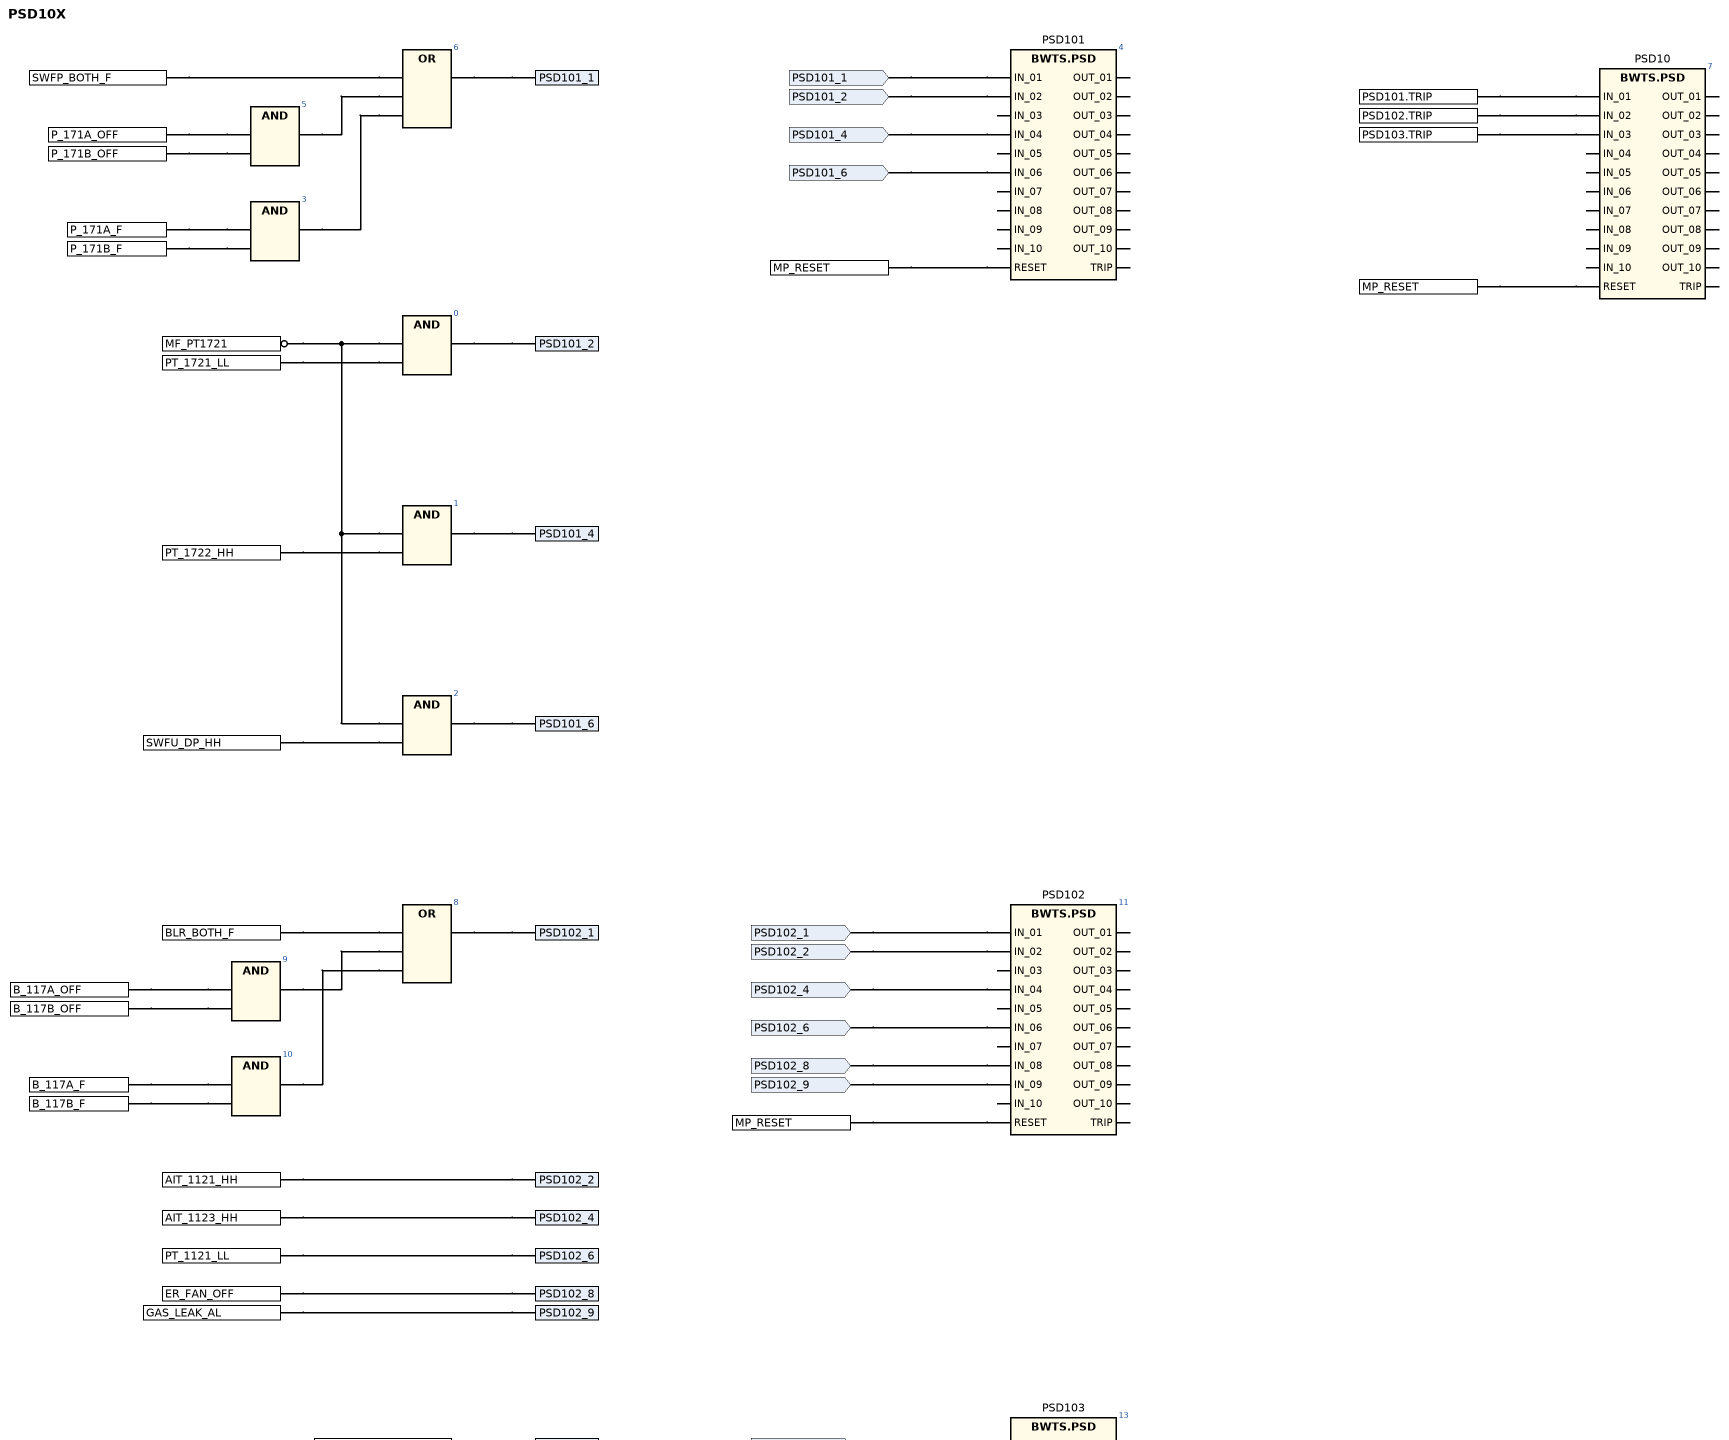
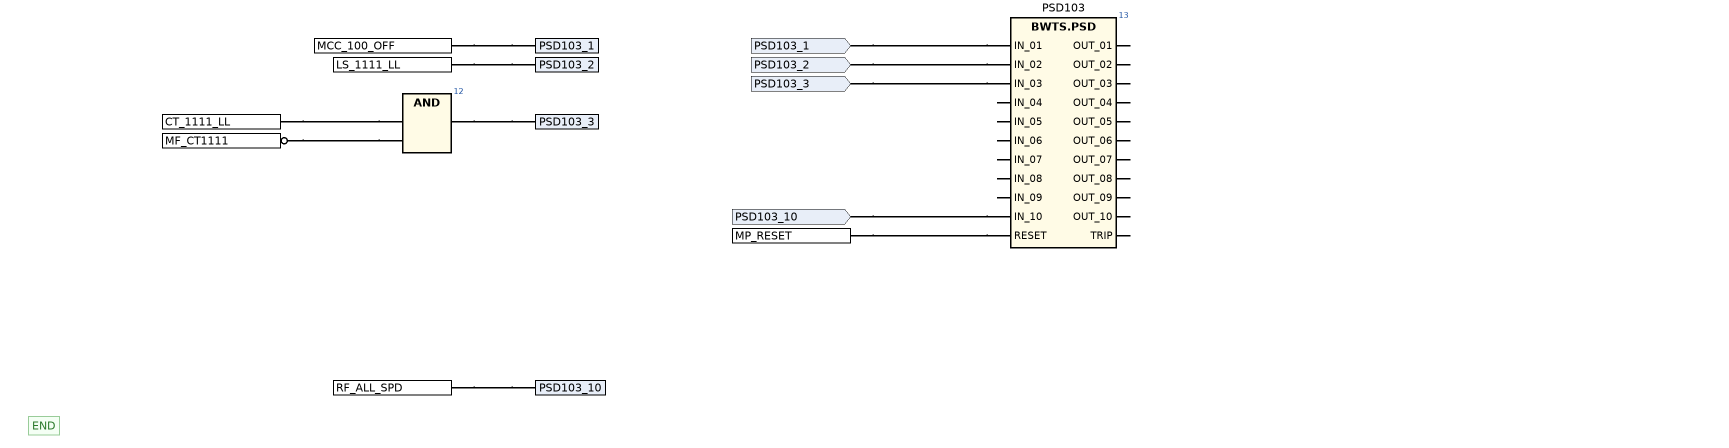
(* NOT MF_PT1721 AND PT_1721_LL; result not used *)
(* NOT MF_PT1721 AND PT_1722_HH; result not used *)
(* NOT MF_PT1721 AND SWFU_DP_HH; result not used *)
_w1 := P_171A_F AND P_171B_F;
PSD101(IN_01 := _w2, IN_02 := _w3, IN_04 := _w4, IN_06 := _w5, RESET := MP_RESET); // BWTS.PSD
(* SWFP_BOTH_F OR P_171A_OFF AND P_171B_OFF OR _w1; result not used *)
PSD10(IN_01 := PSD101.TRIP, IN_02 := PSD102.TRIP, IN_03 := PSD103.TRIP, RESET := MP_RESET); // BWTS.PSD
(* BLR_BOTH_F OR _w6 OR _w7; result not used *)
_w6 := B_117A_OFF AND B_117B_OFF;
_w7 := B_117A_F AND B_117B_F;
PSD102(
    IN_01 := _w8,
    IN_02 := _w9,
    IN_04 := _w10,
    IN_06 := _w11,
    IN_08 := _w12,
    IN_09 := _w13,
    RESET := MP_RESET); // BWTS.PSD
// END
(* CT_1111_LL AND NOT MF_CT1111; result not used *)
PSD103(IN_01 := _w14, IN_02 := _w15, IN_03 := _w16, IN_10 := _w17, RESET := MP_RESET); // BWTS.PSD

END_PROGRAM

// Device/Application/Logic/3.SD/PSD11X
PROGRAM PSD11X
VAR
	
	RS_0: RS;
	TON_0: TON;
END_VAR
VAR // added by the converter: edge detectors and wires of the graphical bodies
    _w1, _w2, _w3, _w4, _w5, _w6, _w7, _w8, _w9, _w10, _w11, _w12, _w13, _w14, _w15, _w16, _w17, _w18, _w19, _w20 : ANY;
END_VAR

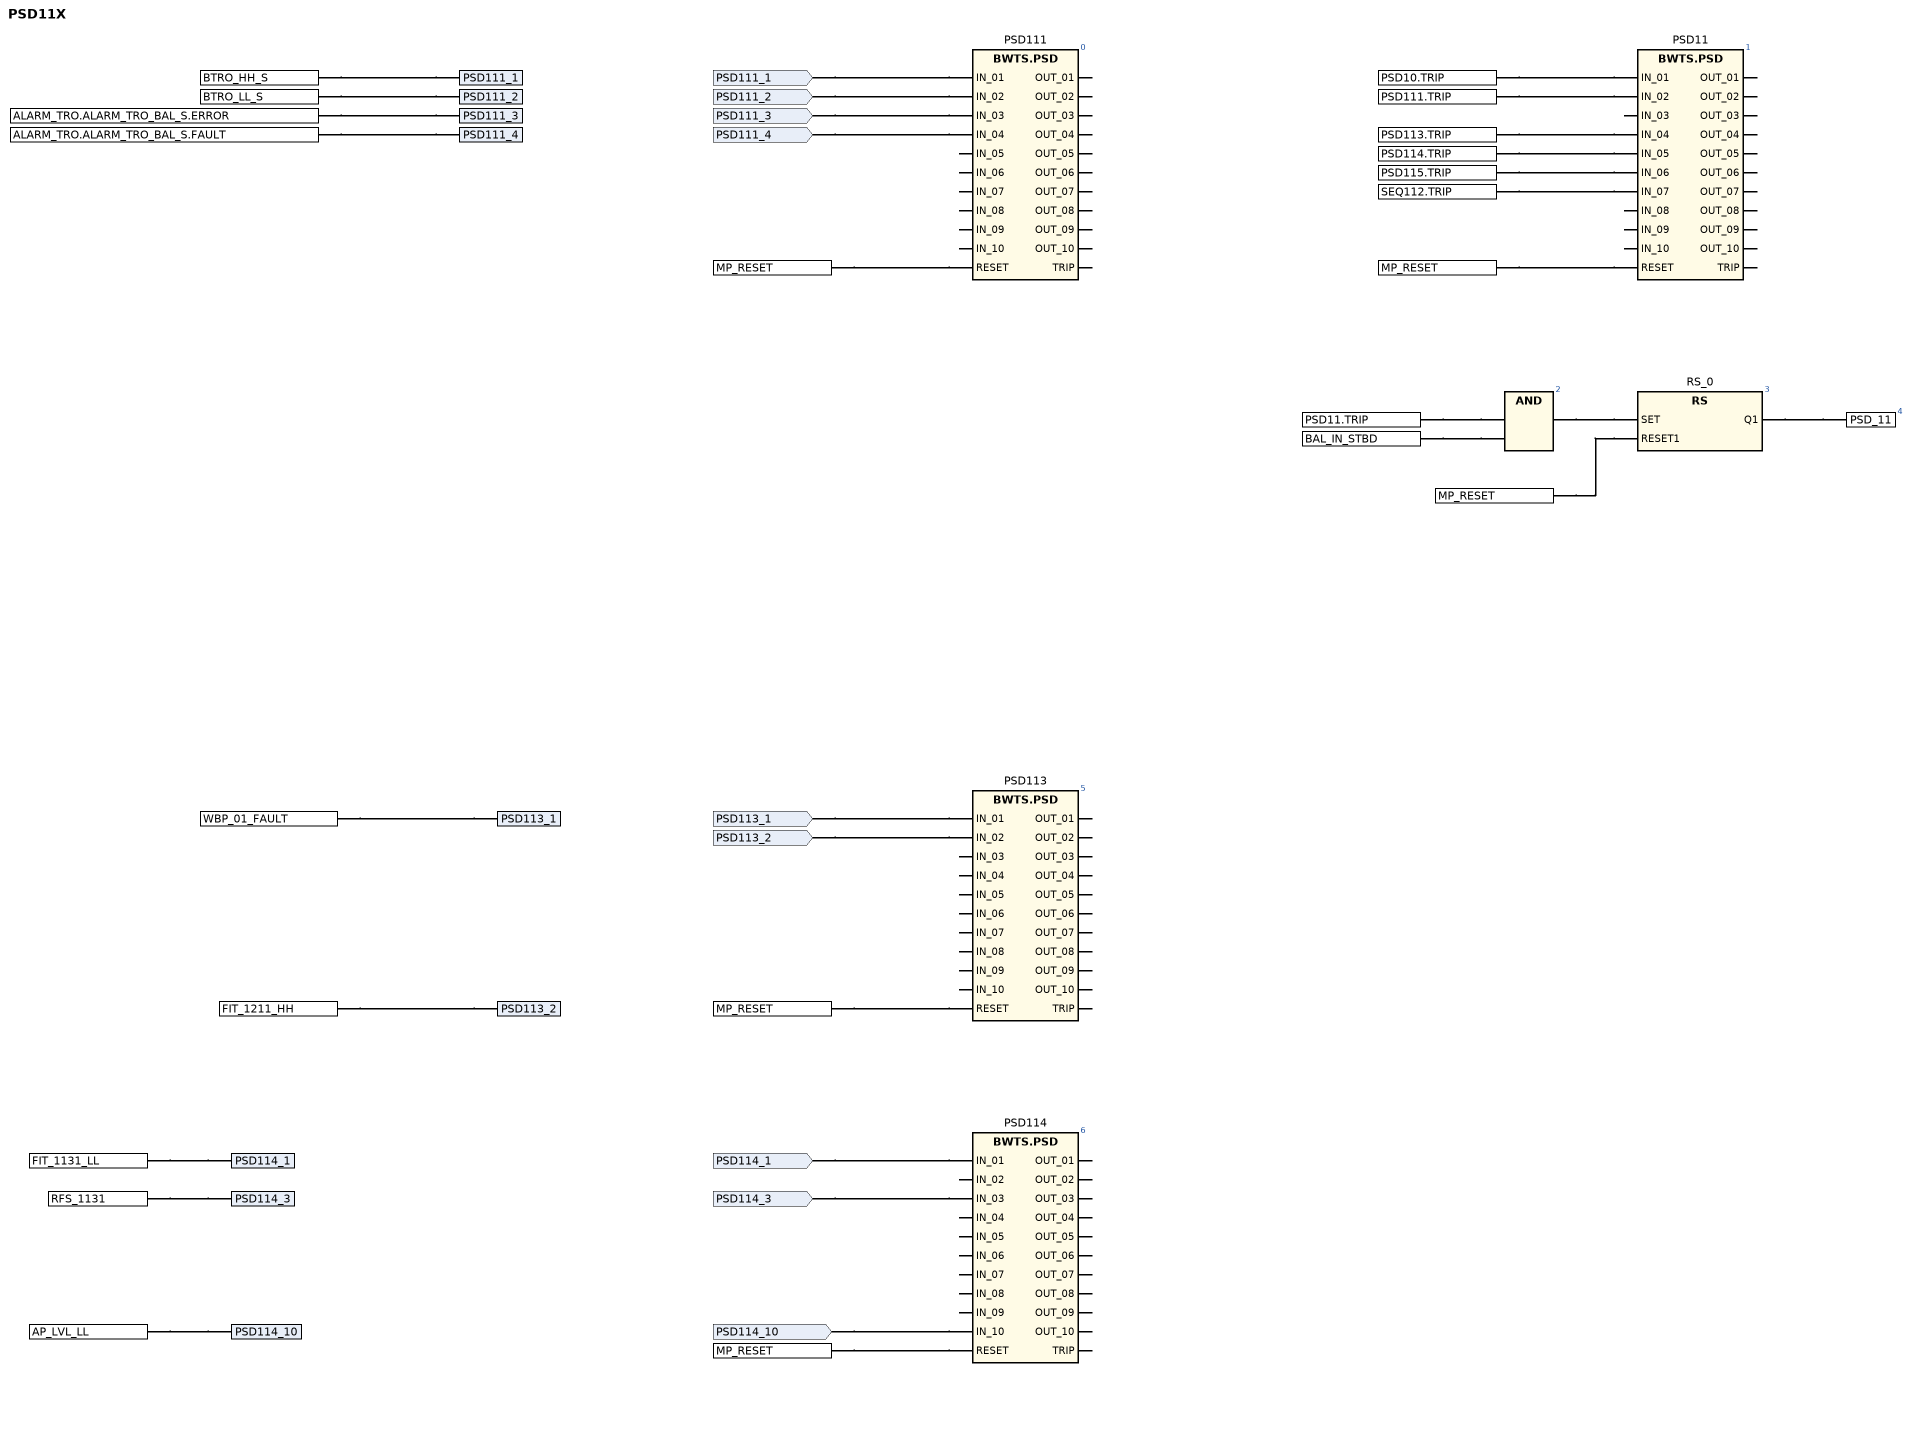
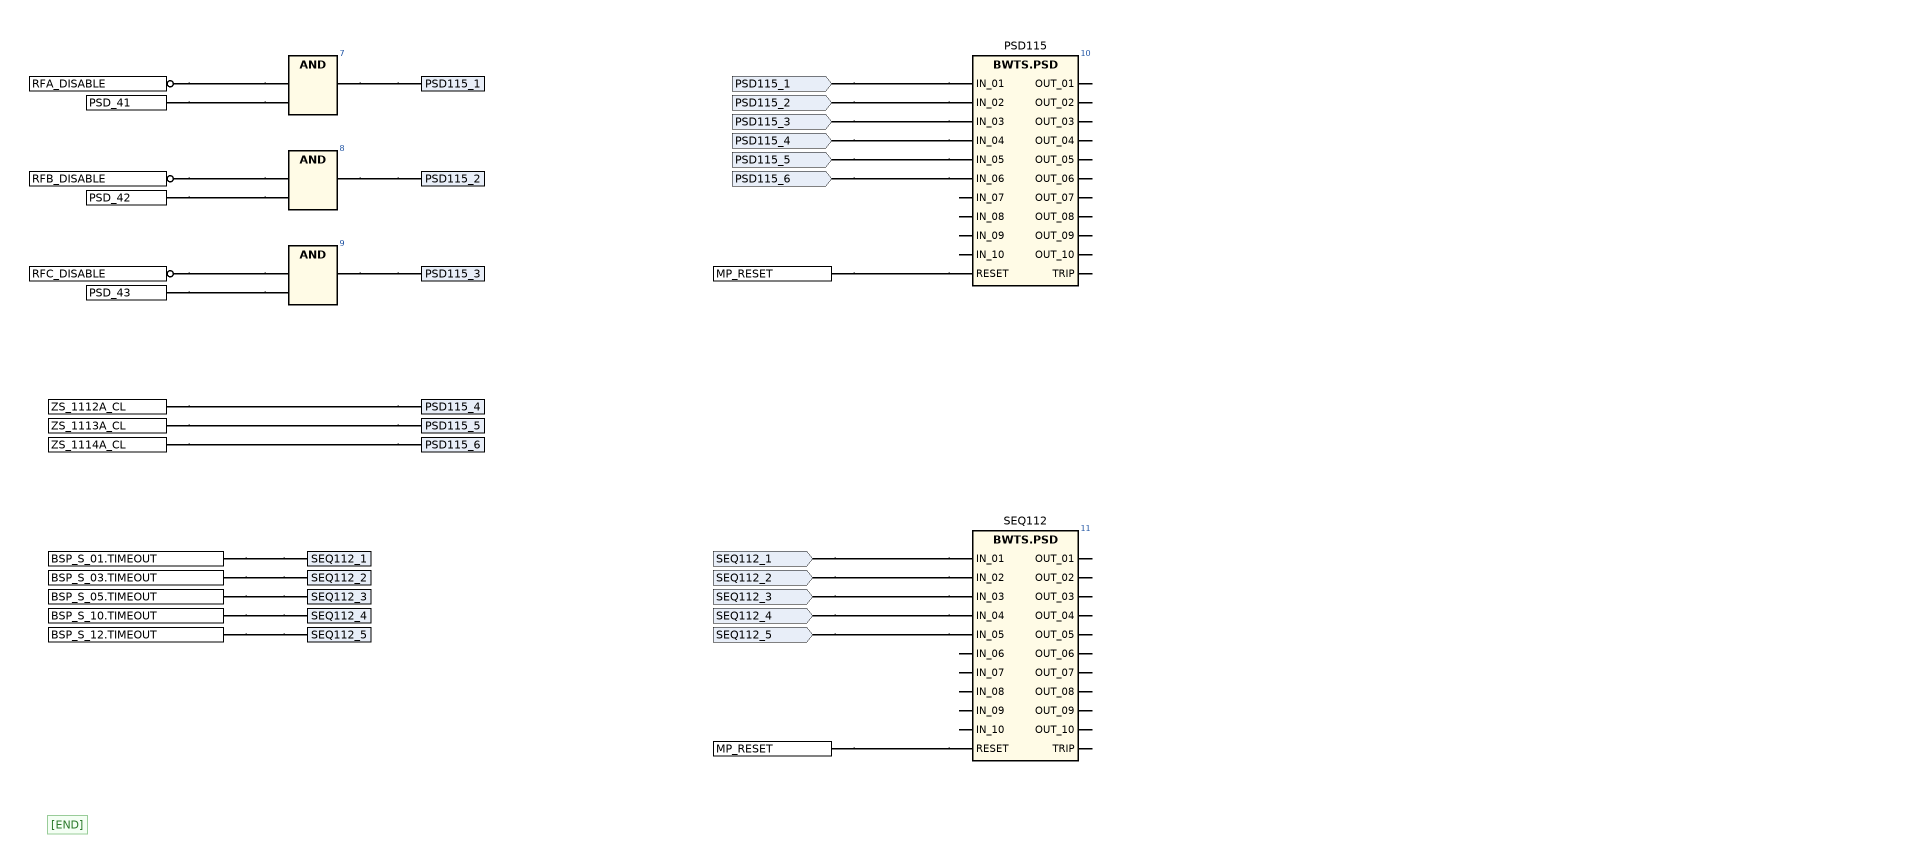
PSD111(IN_01 := _w1, IN_02 := _w2, IN_03 := _w3, IN_04 := _w4, RESET := MP_RESET); // BWTS.PSD
PSD11(
    IN_01 := PSD10.TRIP,
    IN_02 := PSD111.TRIP,
    IN_04 := PSD113.TRIP,
    IN_05 := PSD114.TRIP,
    IN_06 := PSD115.TRIP,
    IN_07 := SEQ112.TRIP,
    RESET := MP_RESET); // BWTS.PSD
RS_0(SET := PSD11.TRIP AND BAL_IN_STBD, RESET1 := MP_RESET); // RS
PSD_11 := RS_0.Q1;
PSD113(IN_01 := _w5, IN_02 := _w6, RESET := MP_RESET); // BWTS.PSD
PSD114(IN_01 := _w7, IN_03 := _w8, IN_10 := _w9, RESET := MP_RESET); // BWTS.PSD
(* NOT RFA_DISABLE AND PSD_41; result not used *)
(* NOT RFB_DISABLE AND PSD_42; result not used *)
(* NOT RFC_DISABLE AND PSD_43; result not used *)
PSD115(
    IN_01 := _w10,
    IN_02 := _w11,
    IN_03 := _w12,
    IN_04 := _w13,
    IN_05 := _w14,
    IN_06 := _w15,
    RESET := MP_RESET); // BWTS.PSD
// [END]
SEQ112(IN_01 := _w16, IN_02 := _w17, IN_03 := _w18, IN_04 := _w19, IN_05 := _w20, RESET := MP_RESET); // BWTS.PSD

END_PROGRAM

// Device/Application/Logic/3.SD/PSD12X
PROGRAM PSD12X
VAR
	
	RS_0: RS;
	TON_0: TON;
END_VAR
VAR // added by the converter: edge detectors and wires of the graphical bodies
    _w1, _w2, _w3, _w4, _w5, _w6, _w7, _w8, _w9, _w10, _w11, _w12, _w13, _w14, _w15, _w16, _w17, _w18, _w19, _w20 : ANY;
END_VAR

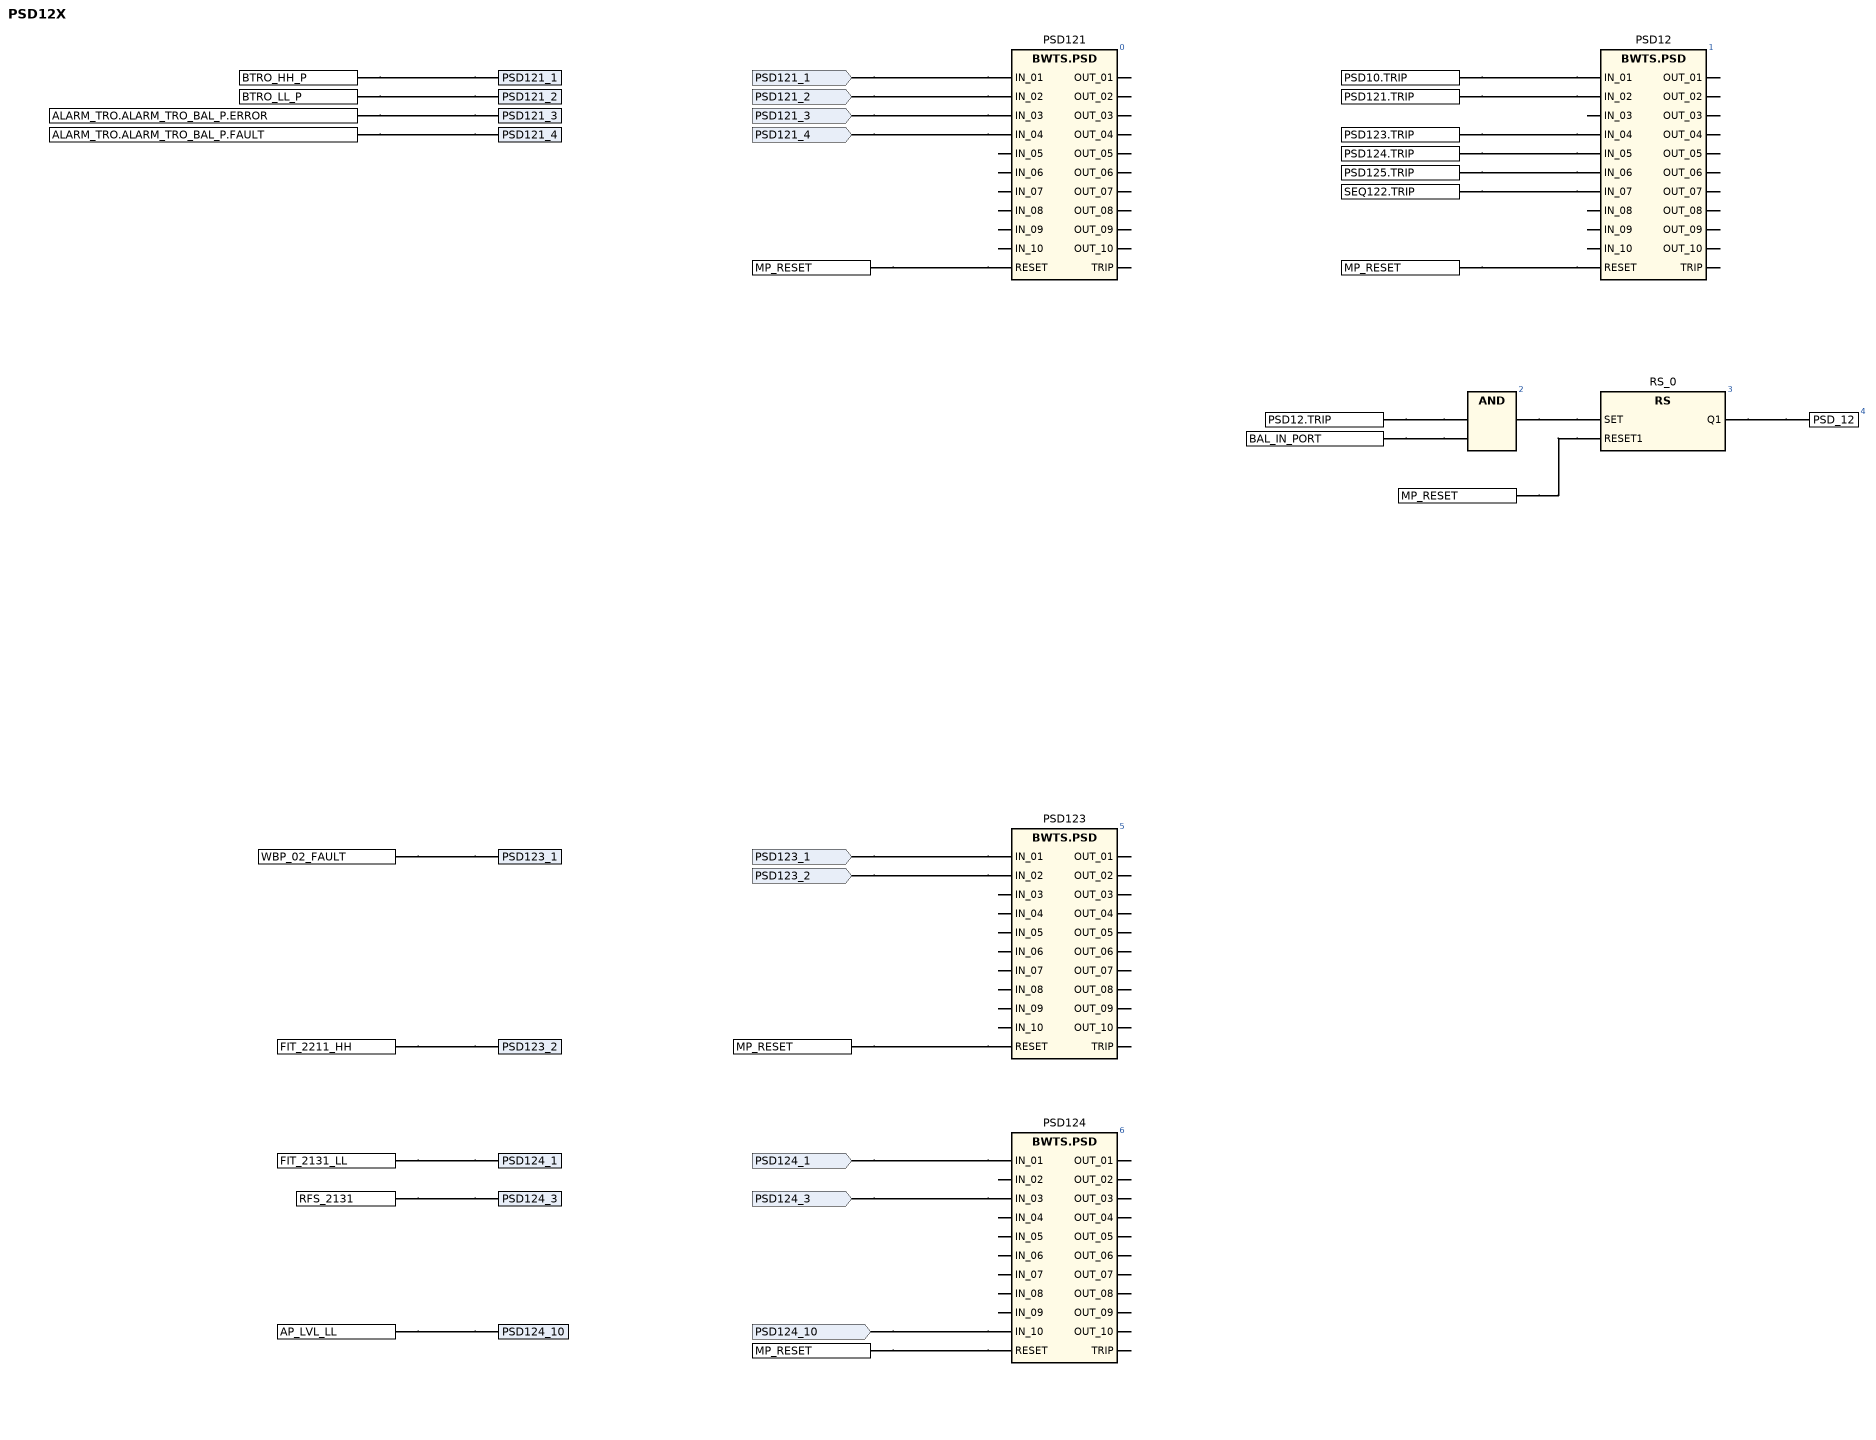
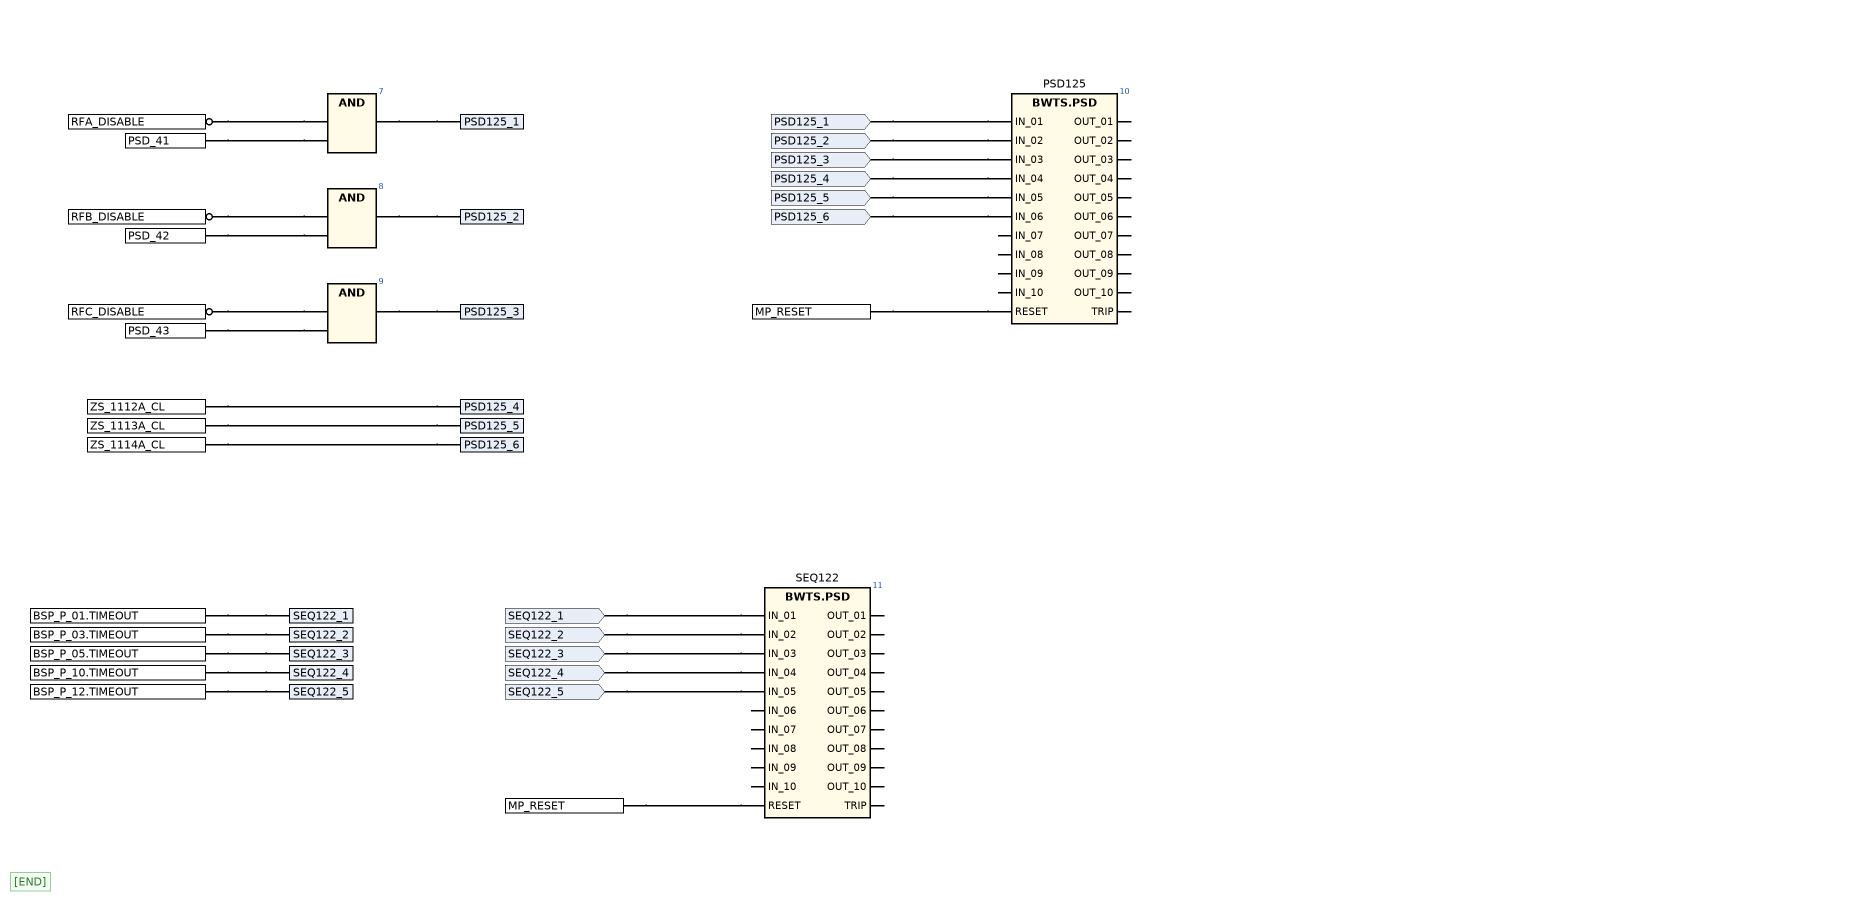
PSD121(IN_01 := _w1, IN_02 := _w2, IN_03 := _w3, IN_04 := _w4, RESET := MP_RESET); // BWTS.PSD
PSD12(
    IN_01 := PSD10.TRIP,
    IN_02 := PSD121.TRIP,
    IN_04 := PSD123.TRIP,
    IN_05 := PSD124.TRIP,
    IN_06 := PSD125.TRIP,
    IN_07 := SEQ122.TRIP,
    RESET := MP_RESET); // BWTS.PSD
RS_0(SET := PSD12.TRIP AND BAL_IN_PORT, RESET1 := MP_RESET); // RS
PSD_12 := RS_0.Q1;
PSD123(IN_01 := _w5, IN_02 := _w6, RESET := MP_RESET); // BWTS.PSD
PSD124(IN_01 := _w7, IN_03 := _w8, IN_10 := _w9, RESET := MP_RESET); // BWTS.PSD
(* NOT RFA_DISABLE AND PSD_41; result not used *)
(* NOT RFB_DISABLE AND PSD_42; result not used *)
(* NOT RFC_DISABLE AND PSD_43; result not used *)
PSD125(
    IN_01 := _w10,
    IN_02 := _w11,
    IN_03 := _w12,
    IN_04 := _w13,
    IN_05 := _w14,
    IN_06 := _w15,
    RESET := MP_RESET); // BWTS.PSD
// [END]
SEQ122(IN_01 := _w16, IN_02 := _w17, IN_03 := _w18, IN_04 := _w19, IN_05 := _w20, RESET := MP_RESET); // BWTS.PSD

END_PROGRAM

// Device/Application/Logic/3.SD/PSD20X
PROGRAM PSD20X
VAR
	
END_VAR
VAR // added by the converter: edge detectors and wires of the graphical bodies
    _w1, _w2, _w3, _w4 : ANY;
END_VAR

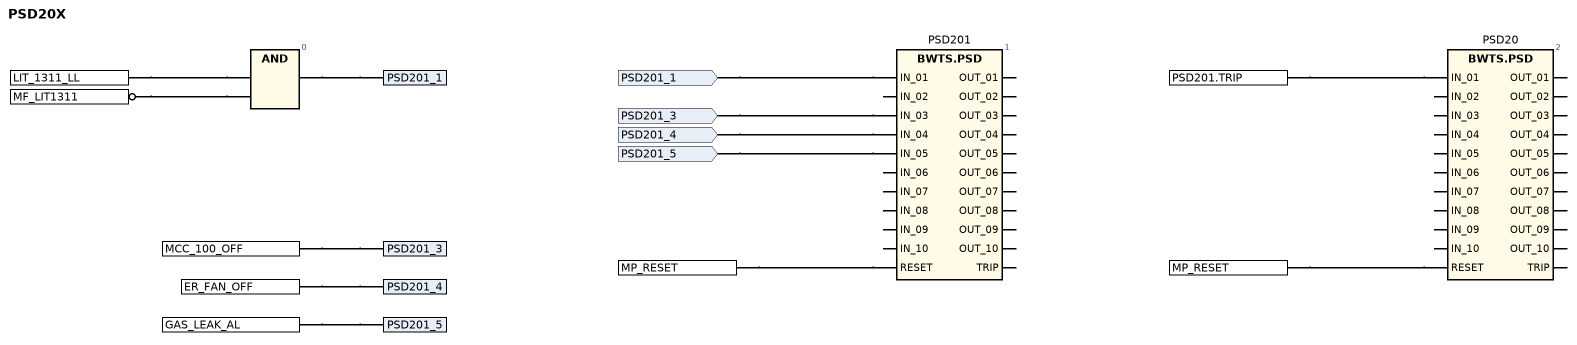
(* LIT_1311_LL AND NOT MF_LIT1311; result not used *)
PSD201(IN_01 := _w1, IN_03 := _w2, IN_04 := _w3, IN_05 := _w4, RESET := MP_RESET); // BWTS.PSD
PSD20(IN_01 := PSD201.TRIP, RESET := MP_RESET); // BWTS.PSD

END_PROGRAM

// Device/Application/Logic/3.SD/PSD21X
PROGRAM PSD21X
VAR
	RS_0: RS;
END_VAR
VAR // added by the converter: edge detectors and wires of the graphical bodies
    _w1, _w2, _w3, _w4, _w5, _w6, _w7, _w8, _w9 : ANY;
END_VAR

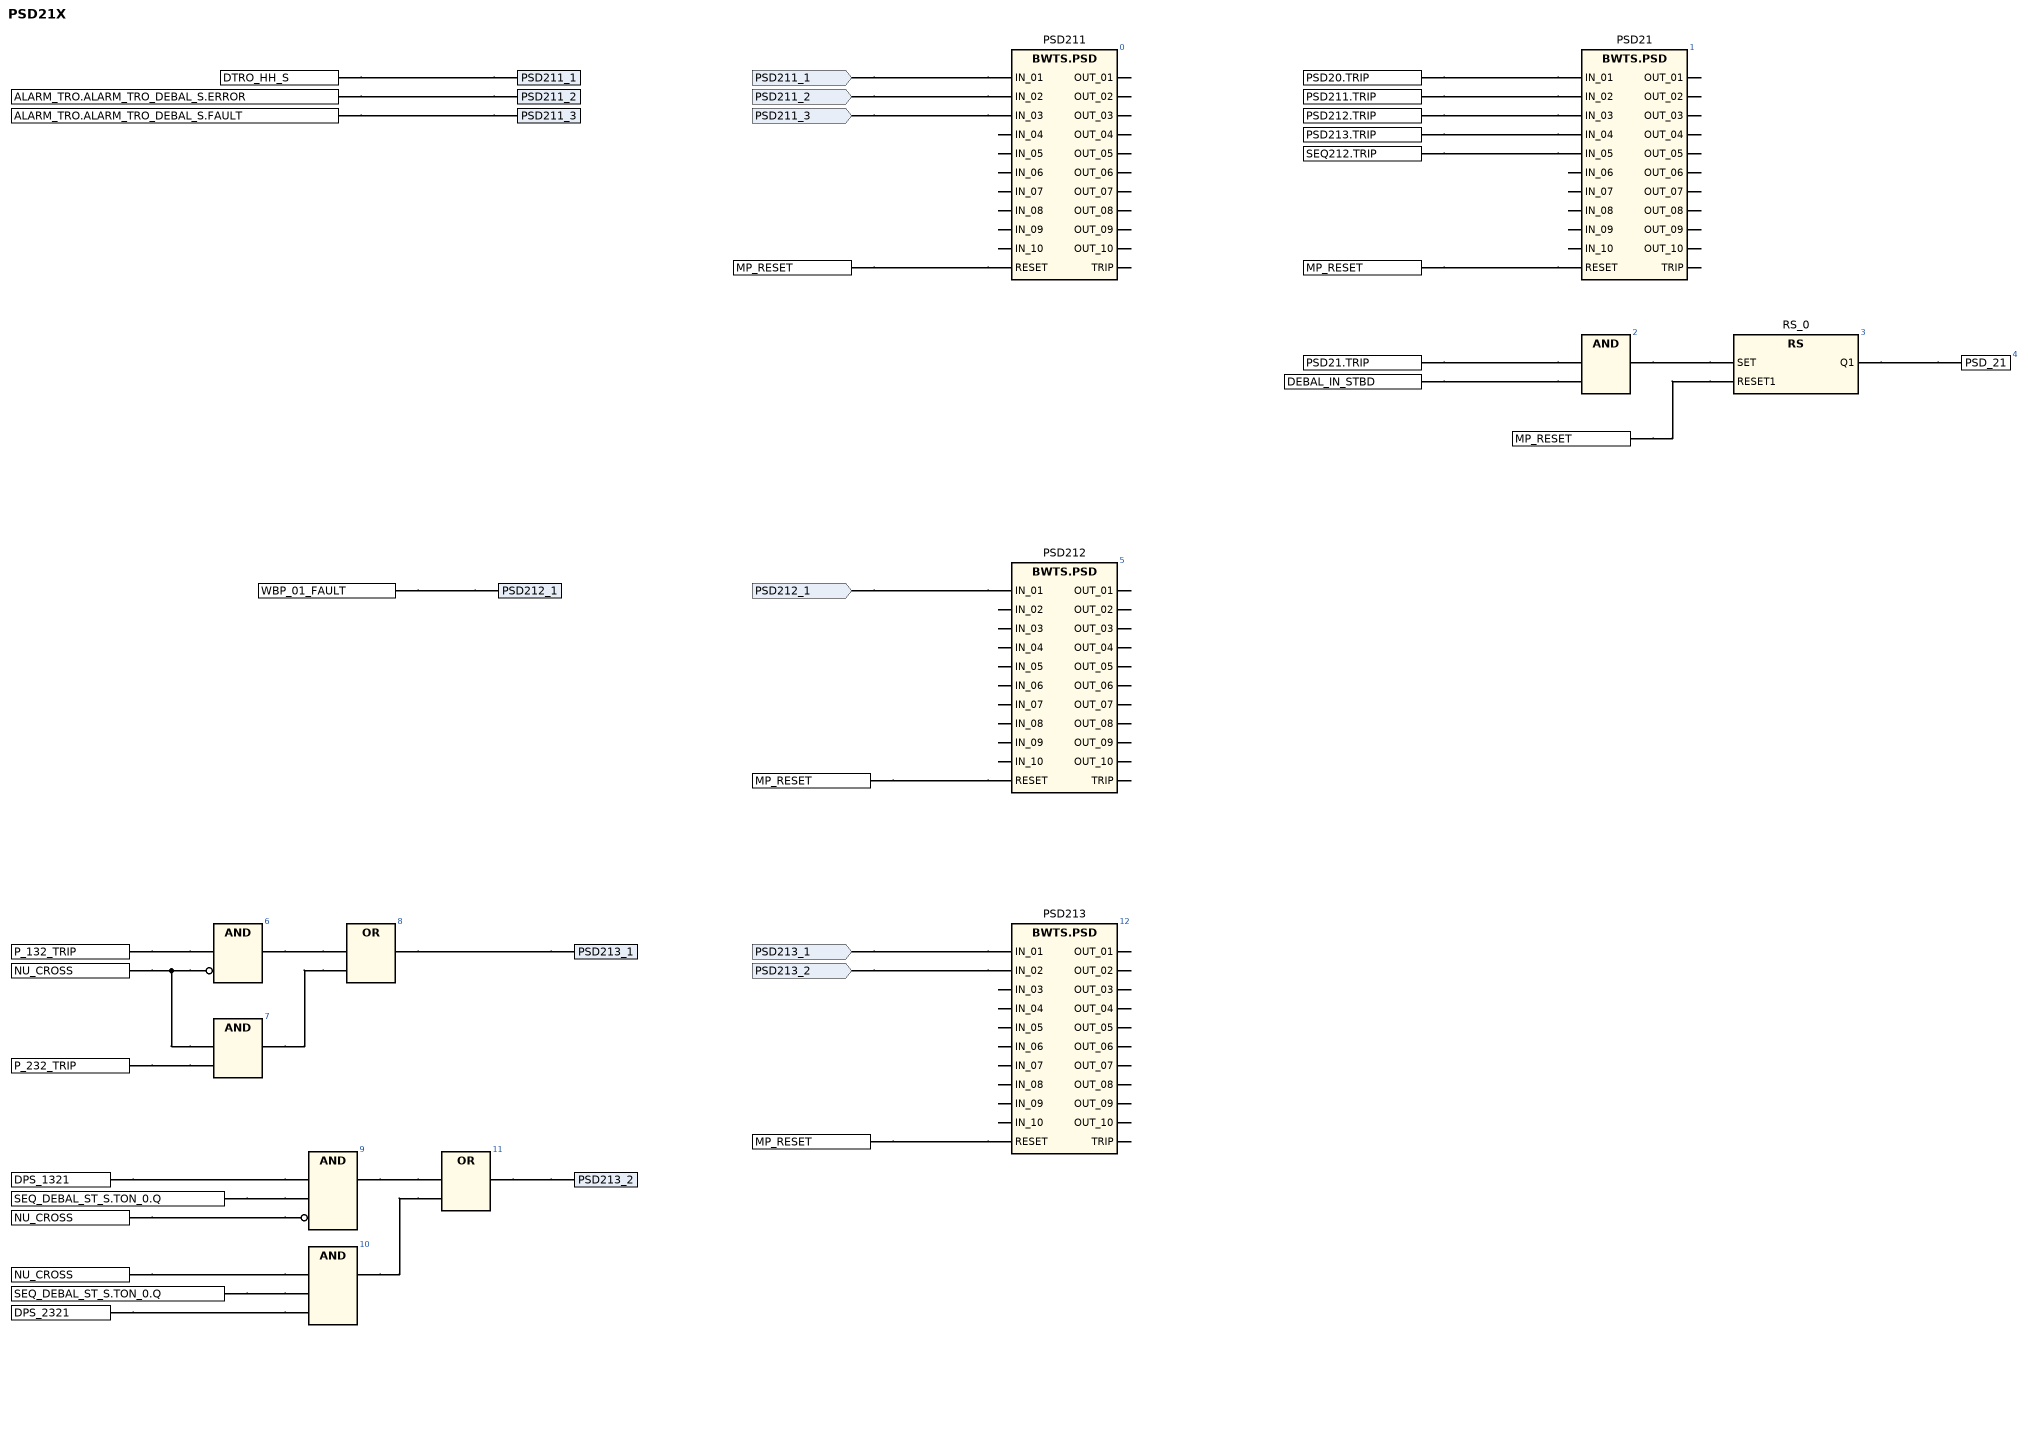
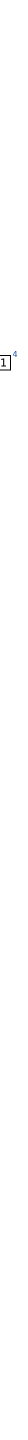
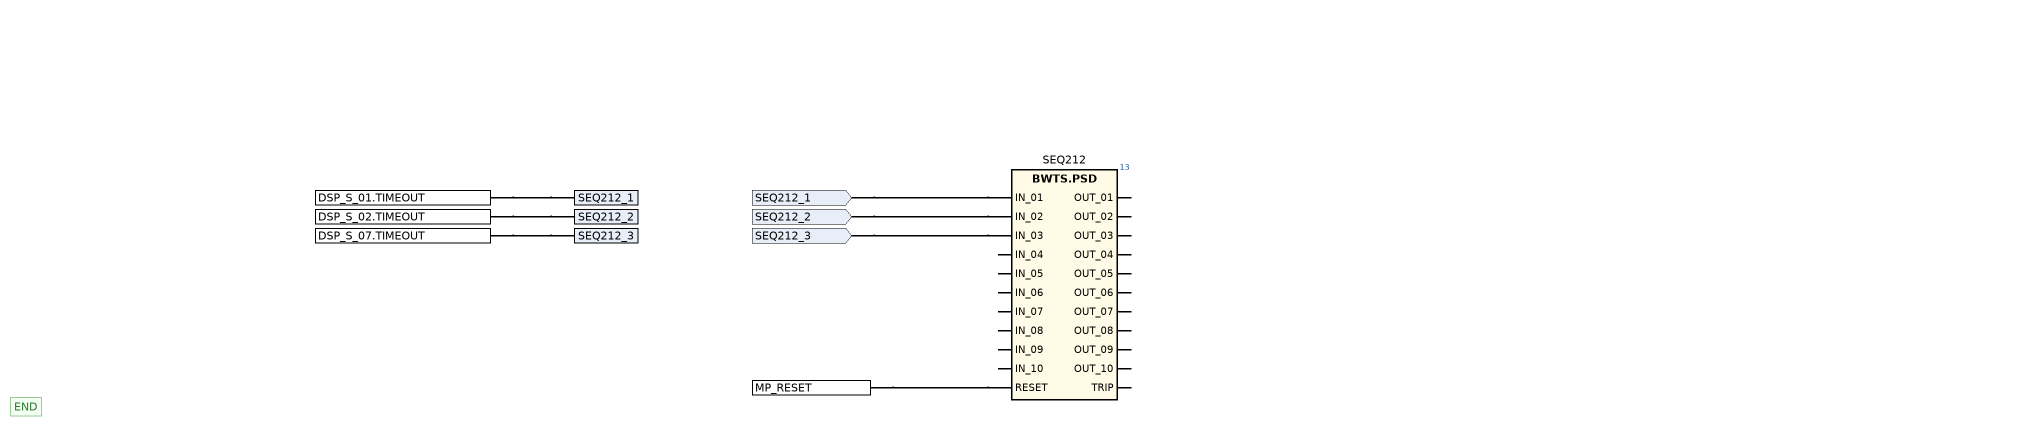
PSD211(IN_01 := _w1, IN_02 := _w2, IN_03 := _w3, RESET := MP_RESET); // BWTS.PSD
PSD21(
    IN_01 := PSD20.TRIP,
    IN_02 := PSD211.TRIP,
    IN_03 := PSD212.TRIP,
    IN_04 := PSD213.TRIP,
    IN_05 := SEQ212.TRIP,
    RESET := MP_RESET); // BWTS.PSD
RS_0(SET := PSD21.TRIP AND DEBAL_IN_STBD, RESET1 := MP_RESET); // RS
PSD_21 := RS_0.Q1;
PSD212(IN_01 := _w4, RESET := MP_RESET); // BWTS.PSD
(* P_132_TRIP AND NOT NU_CROSS OR NU_CROSS AND P_232_TRIP; result not used *)
(* DPS_1321 AND SEQ_DEBAL_ST_S.TON_0.Q AND NOT NU_CROSS OR NU_CROSS AND SEQ_DEBAL_ST_S.TON_0.Q AND DPS_2321; result not used *)
PSD213(IN_01 := _w5, IN_02 := _w6, RESET := MP_RESET); // BWTS.PSD
// END
SEQ212(IN_01 := _w7, IN_02 := _w8, IN_03 := _w9, RESET := MP_RESET); // BWTS.PSD

END_PROGRAM

// Device/Application/Logic/3.SD/PSD22X
PROGRAM PSD22X
VAR
	RS_0: RS;
END_VAR
VAR // added by the converter: edge detectors and wires of the graphical bodies
    _w1, _w3, _w4, _w5, _w8, _w9, _w10, _w11, _w12, _w13 : ANY;
    _w2, _w6, _w7 : BOOL;
END_VAR

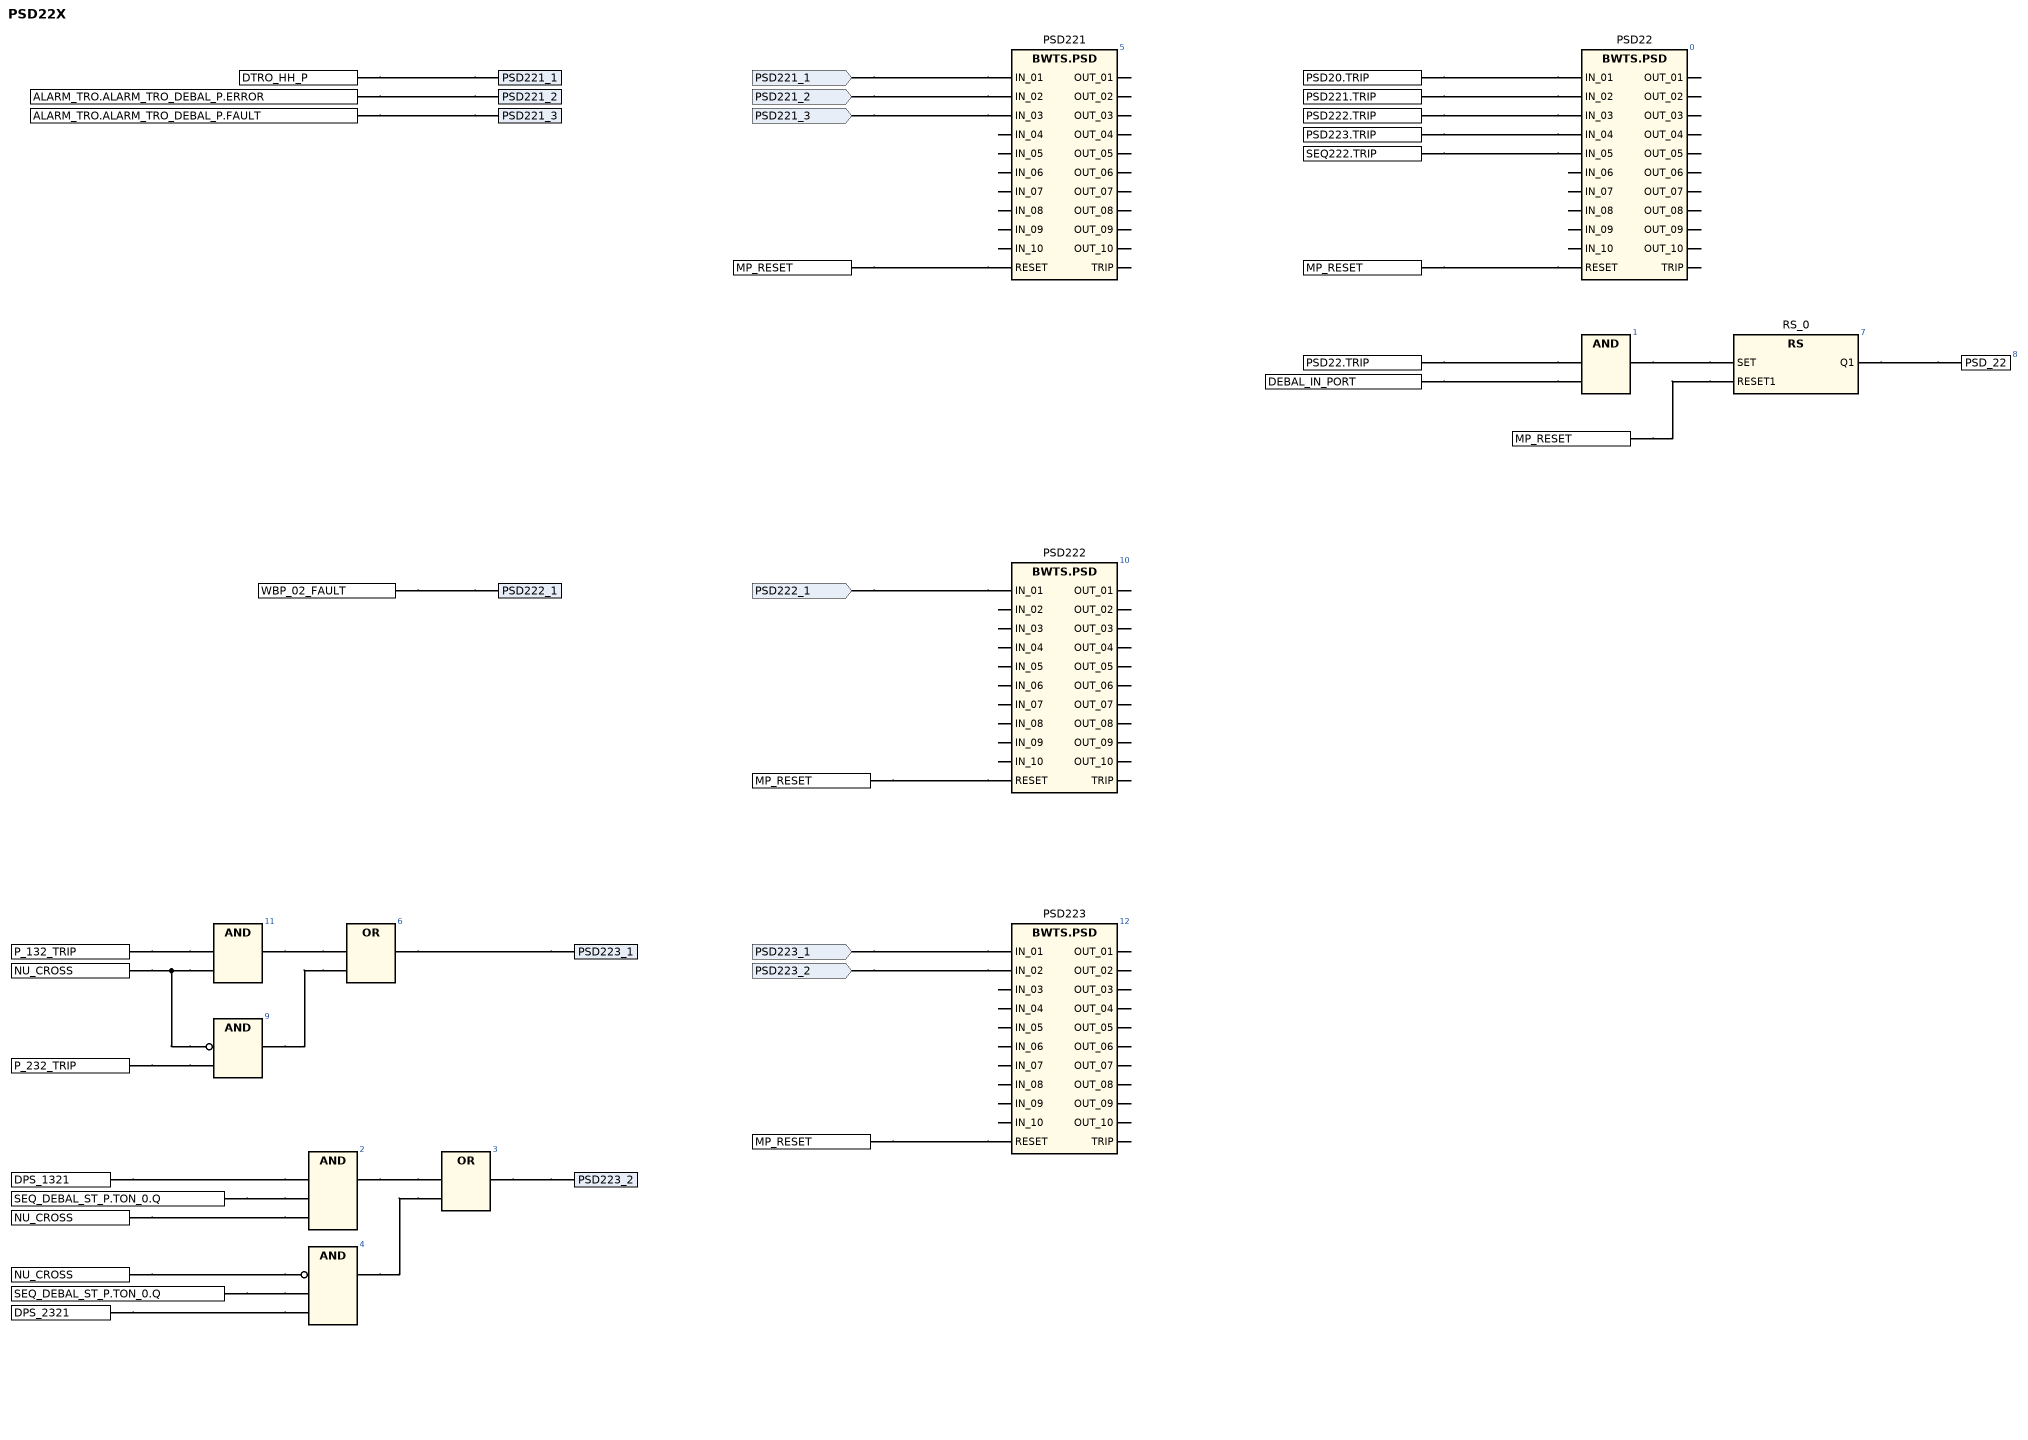
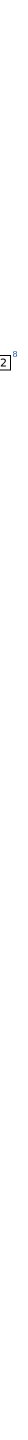
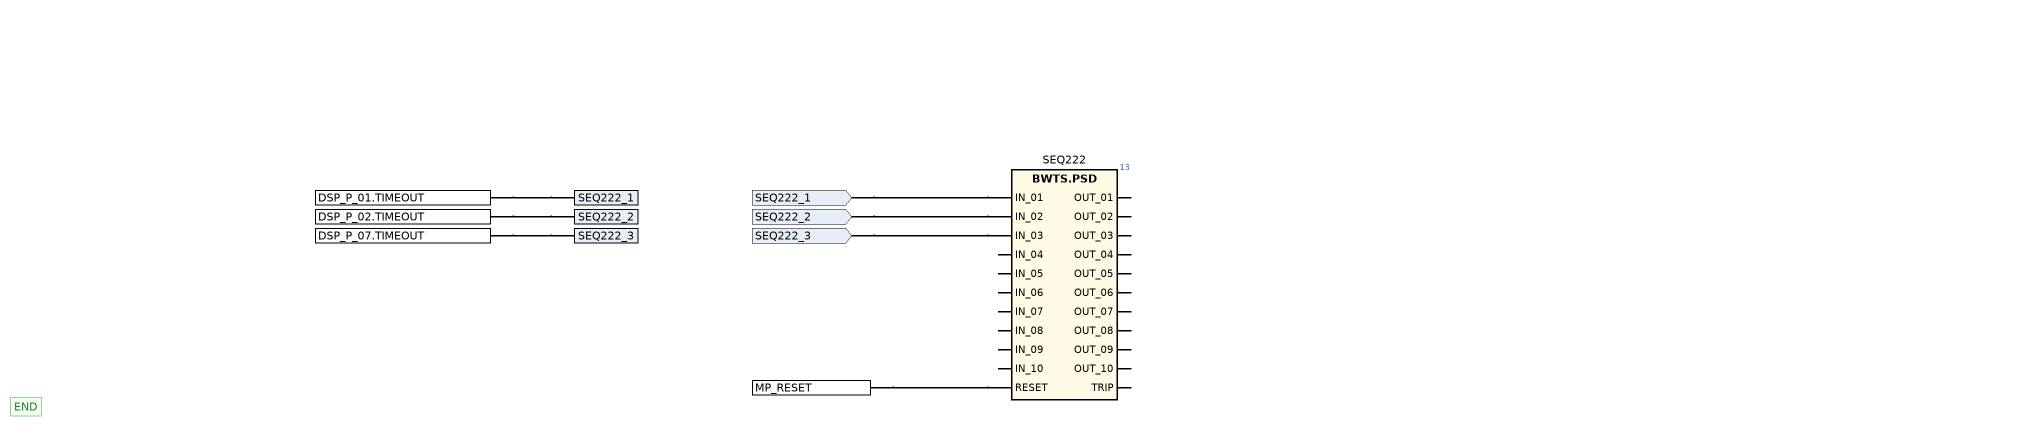
PSD22(
    IN_01 := PSD20.TRIP,
    IN_02 := PSD221.TRIP,
    IN_03 := PSD222.TRIP,
    IN_04 := PSD223.TRIP,
    IN_05 := SEQ222.TRIP,
    RESET := MP_RESET); // BWTS.PSD
_w1 := PSD22.TRIP AND DEBAL_IN_PORT;
(* DPS_1321 AND SEQ_DEBAL_ST_P.TON_0.Q AND NU_CROSS OR _w2; result not used *)
_w2 := NOT NU_CROSS AND SEQ_DEBAL_ST_P.TON_0.Q AND DPS_2321;
PSD221(IN_01 := _w3, IN_02 := _w4, IN_03 := _w5, RESET := MP_RESET); // BWTS.PSD
(* _w6 OR _w7; result not used *)
RS_0(SET := _w1, RESET1 := MP_RESET); // RS
PSD_22 := RS_0.Q1;
_w7 := NOT NU_CROSS AND P_232_TRIP;
PSD222(IN_01 := _w8, RESET := MP_RESET); // BWTS.PSD
_w6 := P_132_TRIP AND NU_CROSS;
PSD223(IN_01 := _w9, IN_02 := _w10, RESET := MP_RESET); // BWTS.PSD
// END
SEQ222(IN_01 := _w11, IN_02 := _w12, IN_03 := _w13, RESET := MP_RESET); // BWTS.PSD

END_PROGRAM

// Device/Application/Logic/3.SD/PSD30X
PROGRAM PSD30X
VAR
	
END_VAR
VAR // added by the converter: edge detectors and wires of the graphical bodies
    _w1, _w2, _w3, _w4 : ANY;
END_VAR

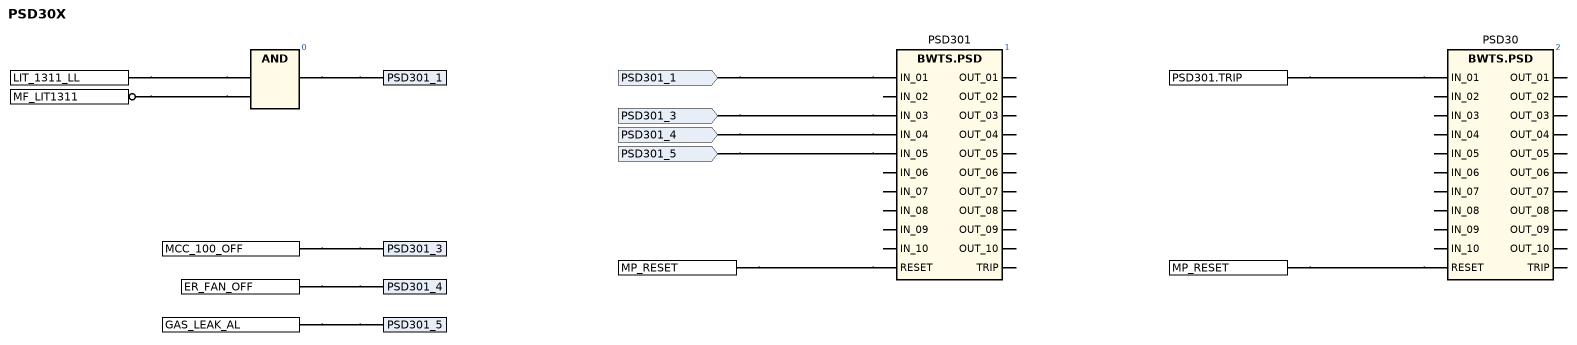
(* LIT_1311_LL AND NOT MF_LIT1311; result not used *)
PSD301(IN_01 := _w1, IN_03 := _w2, IN_04 := _w3, IN_05 := _w4, RESET := MP_RESET); // BWTS.PSD
PSD30(IN_01 := PSD301.TRIP, RESET := MP_RESET); // BWTS.PSD

END_PROGRAM

// Device/Application/Logic/3.SD/PSD31X
PROGRAM PSD31X
VAR
	RS_0: RS;
END_VAR
VAR // added by the converter: edge detectors and wires of the graphical bodies
    _w1, _w2, _w3, _w4, _w5, _w6, _w7, _w8, _w9 : ANY;
END_VAR

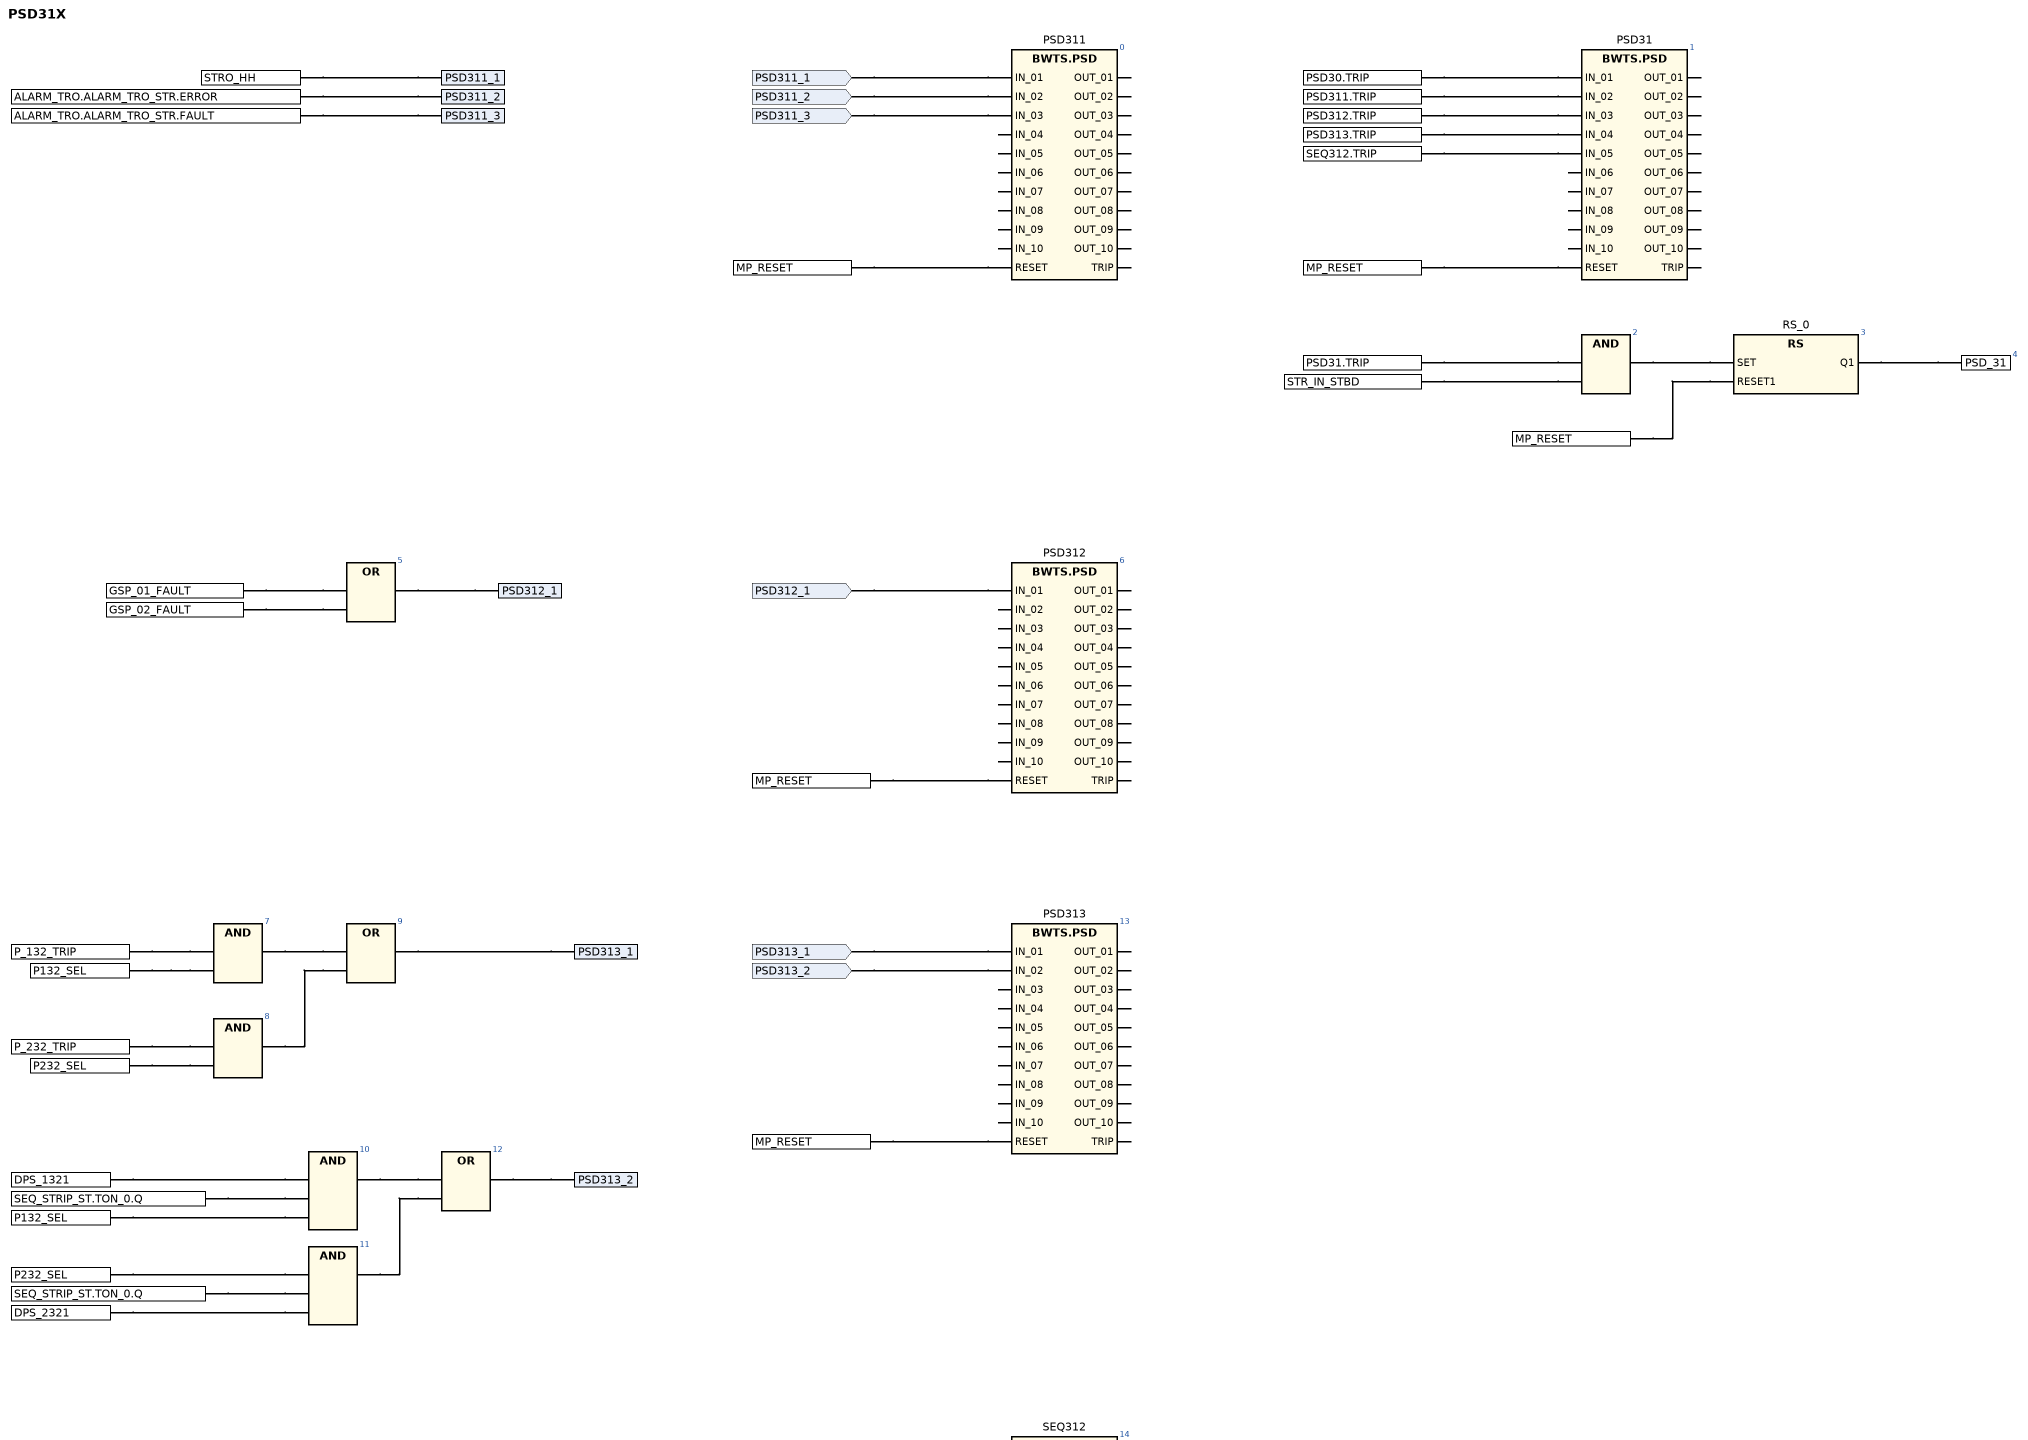
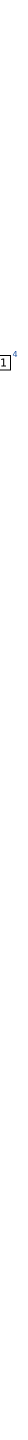
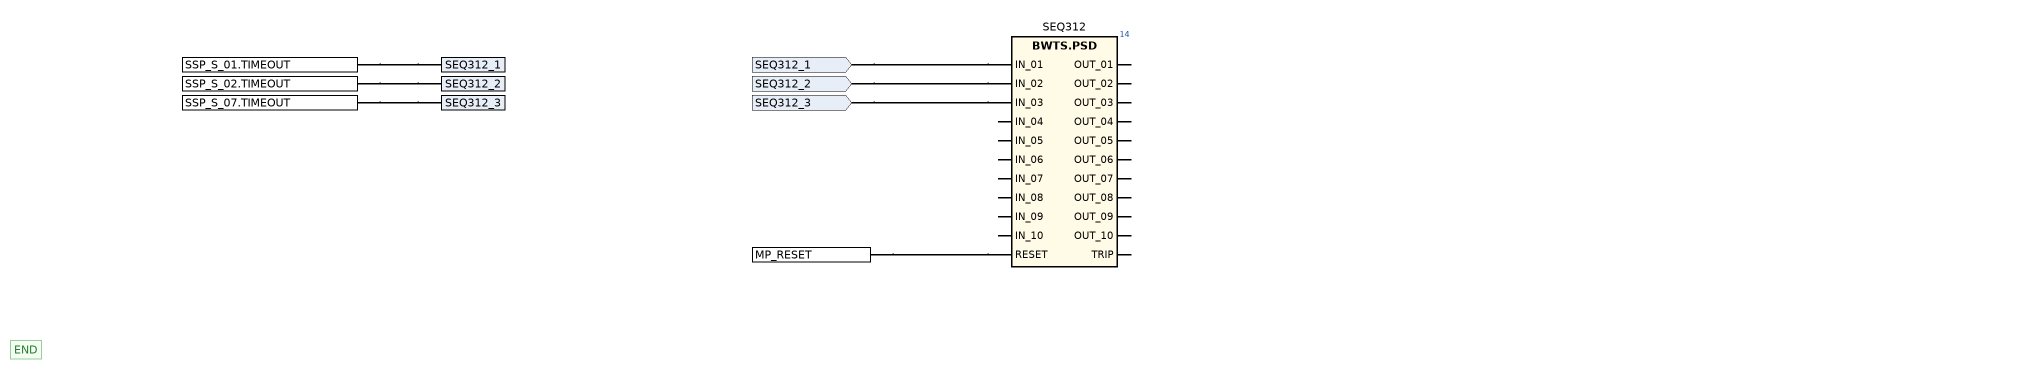
PSD311(IN_01 := _w1, IN_02 := _w2, IN_03 := _w3, RESET := MP_RESET); // BWTS.PSD
PSD31(
    IN_01 := PSD30.TRIP,
    IN_02 := PSD311.TRIP,
    IN_03 := PSD312.TRIP,
    IN_04 := PSD313.TRIP,
    IN_05 := SEQ312.TRIP,
    RESET := MP_RESET); // BWTS.PSD
RS_0(SET := PSD31.TRIP AND STR_IN_STBD, RESET1 := MP_RESET); // RS
PSD_31 := RS_0.Q1;
(* GSP_01_FAULT OR GSP_02_FAULT; result not used *)
PSD312(IN_01 := _w4, RESET := MP_RESET); // BWTS.PSD
(* P_132_TRIP AND P132_SEL OR P_232_TRIP AND P232_SEL; result not used *)
(* DPS_1321 AND SEQ_STRIP_ST.TON_0.Q AND P132_SEL OR P232_SEL AND SEQ_STRIP_ST.TON_0.Q AND DPS_2321; result not used *)
PSD313(IN_01 := _w5, IN_02 := _w6, RESET := MP_RESET); // BWTS.PSD
// END
SEQ312(IN_01 := _w7, IN_02 := _w8, IN_03 := _w9, RESET := MP_RESET); // BWTS.PSD

END_PROGRAM

// Device/Application/Logic/3.SD/USD41X
PROGRAM USD41X
VAR

END_VAR
VAR // added by the converter: edge detectors and wires of the graphical bodies
    _w1, _w2, _w3, _w4 : ANY;
END_VAR

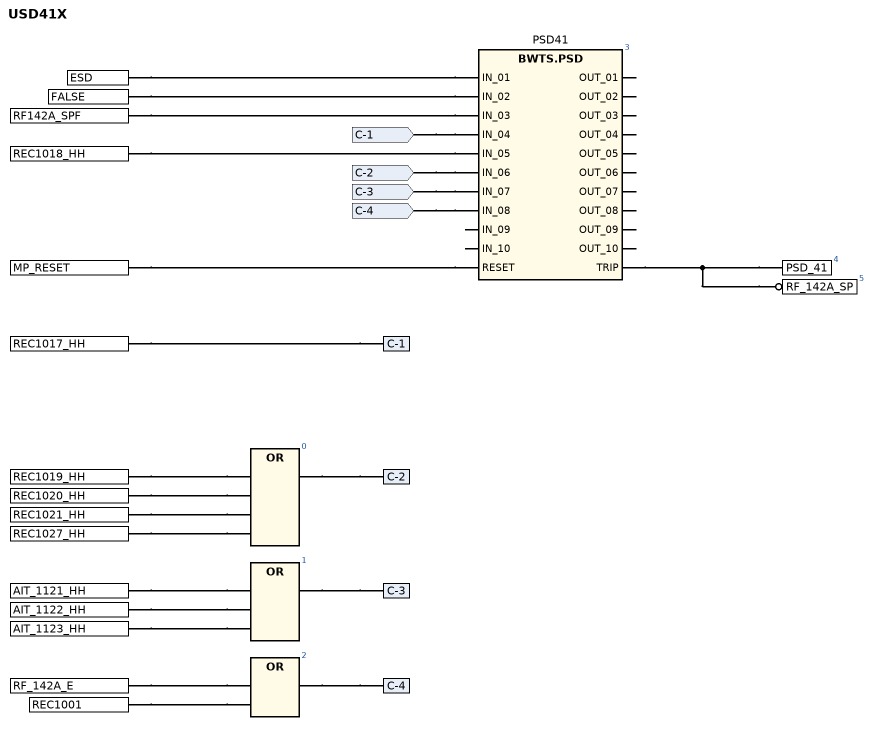
(* REC1019_HH OR REC1020_HH OR REC1021_HH OR REC1027_HH; result not used *)
(* AIT_1121_HH OR AIT_1122_HH OR AIT_1123_HH; result not used *)
(* RF_142A_E OR REC1001; result not used *)
PSD41(
    IN_01 := ESD,
    IN_02 := FALSE,
    IN_03 := RF142A_SPF,
    IN_04 := _w1,
    IN_05 := REC1018_HH,
    IN_06 := _w2,
    IN_07 := _w3,
    IN_08 := _w4,
    RESET := MP_RESET); // BWTS.PSD
PSD_41 := PSD41.TRIP;
RF_142A_SP := NOT PSD41.TRIP;

END_PROGRAM

// Device/Application/Logic/3.SD/USD42X
PROGRAM USD42X
VAR

END_VAR
VAR // added by the converter: edge detectors and wires of the graphical bodies
    _w1, _w2, _w3, _w4 : ANY;
END_VAR

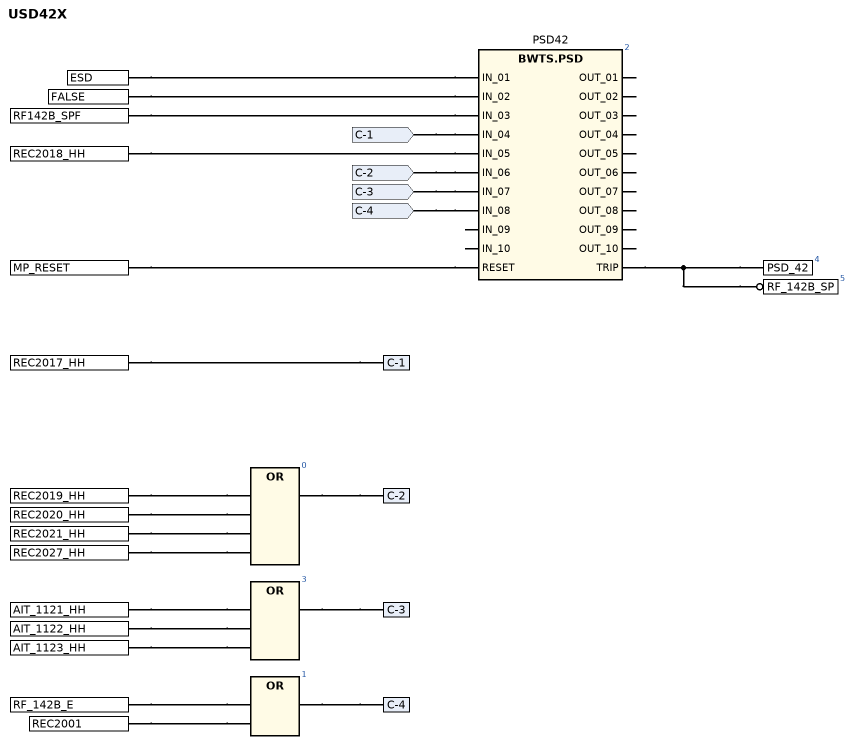
(* REC2019_HH OR REC2020_HH OR REC2021_HH OR REC2027_HH; result not used *)
(* RF_142B_E OR REC2001; result not used *)
PSD42(
    IN_01 := ESD,
    IN_02 := FALSE,
    IN_03 := RF142B_SPF,
    IN_04 := _w1,
    IN_05 := REC2018_HH,
    IN_06 := _w2,
    IN_07 := _w3,
    IN_08 := _w4,
    RESET := MP_RESET); // BWTS.PSD
(* AIT_1121_HH OR AIT_1122_HH OR AIT_1123_HH; result not used *)
PSD_42 := PSD42.TRIP;
RF_142B_SP := NOT PSD42.TRIP;

END_PROGRAM

// Device/Application/Logic/3.SD/USD43X
PROGRAM USD43X
VAR

END_VAR
VAR // added by the converter: edge detectors and wires of the graphical bodies
    _w1, _w2, _w3, _w4 : ANY;
END_VAR

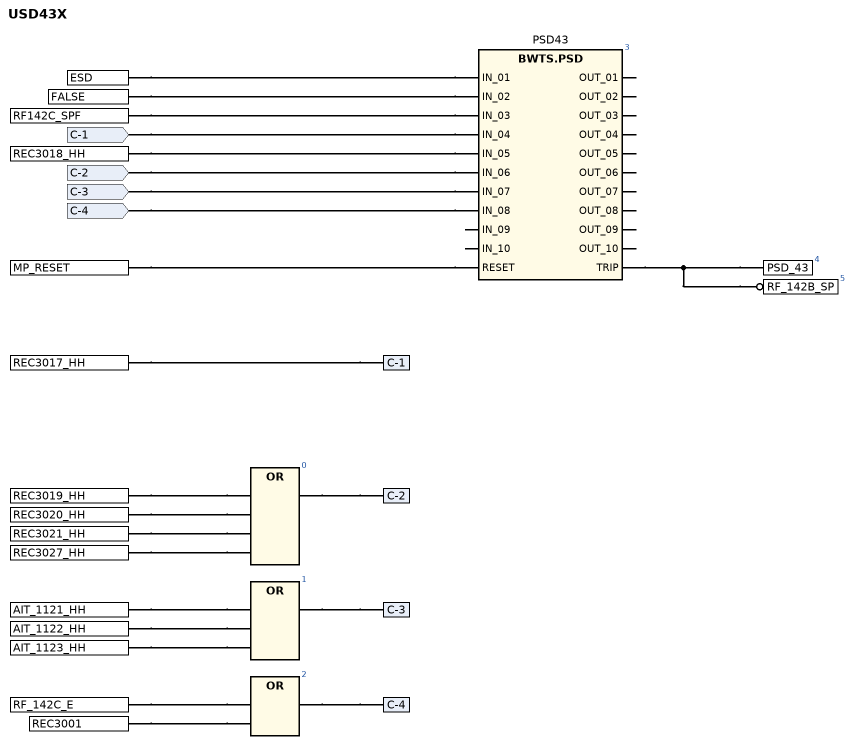
(* REC3019_HH OR REC3020_HH OR REC3021_HH OR REC3027_HH; result not used *)
(* AIT_1121_HH OR AIT_1122_HH OR AIT_1123_HH; result not used *)
(* RF_142C_E OR REC3001; result not used *)
PSD43(
    IN_01 := ESD,
    IN_02 := FALSE,
    IN_03 := RF142C_SPF,
    IN_04 := _w1,
    IN_05 := REC3018_HH,
    IN_06 := _w2,
    IN_07 := _w3,
    IN_08 := _w4,
    RESET := MP_RESET); // BWTS.PSD
PSD_43 := PSD43.TRIP;
RF_142B_SP := NOT PSD43.TRIP;

END_PROGRAM

// Device/Application/Logic/0.SIMULATION/SCENARIO
PROGRAM SCENARIO
VAR
	RS_SCEN1: RS;
	RS_SCEN2_1: RS;
	RS_SCEN2_2: RS;
	RS_SCEN3_1: RS;
	RS_SCEN3_2: RS;
	RS_SCEN4_1: RS;
	RS_SCEN4_2: RS;
	RS_SCEN5: RS;
	RS_SCEN6: RS;
	RS_SCEN7: RS;
	RS_SCEN8_1: RS;
	RS_SCEN8_2: RS;
	RS_SCEN9_1: RS;
	RS_SCEN9_2: RS;
	RS_SCEN10_1: RS;
	RS_SCEN10_2: RS;
	
END_VAR

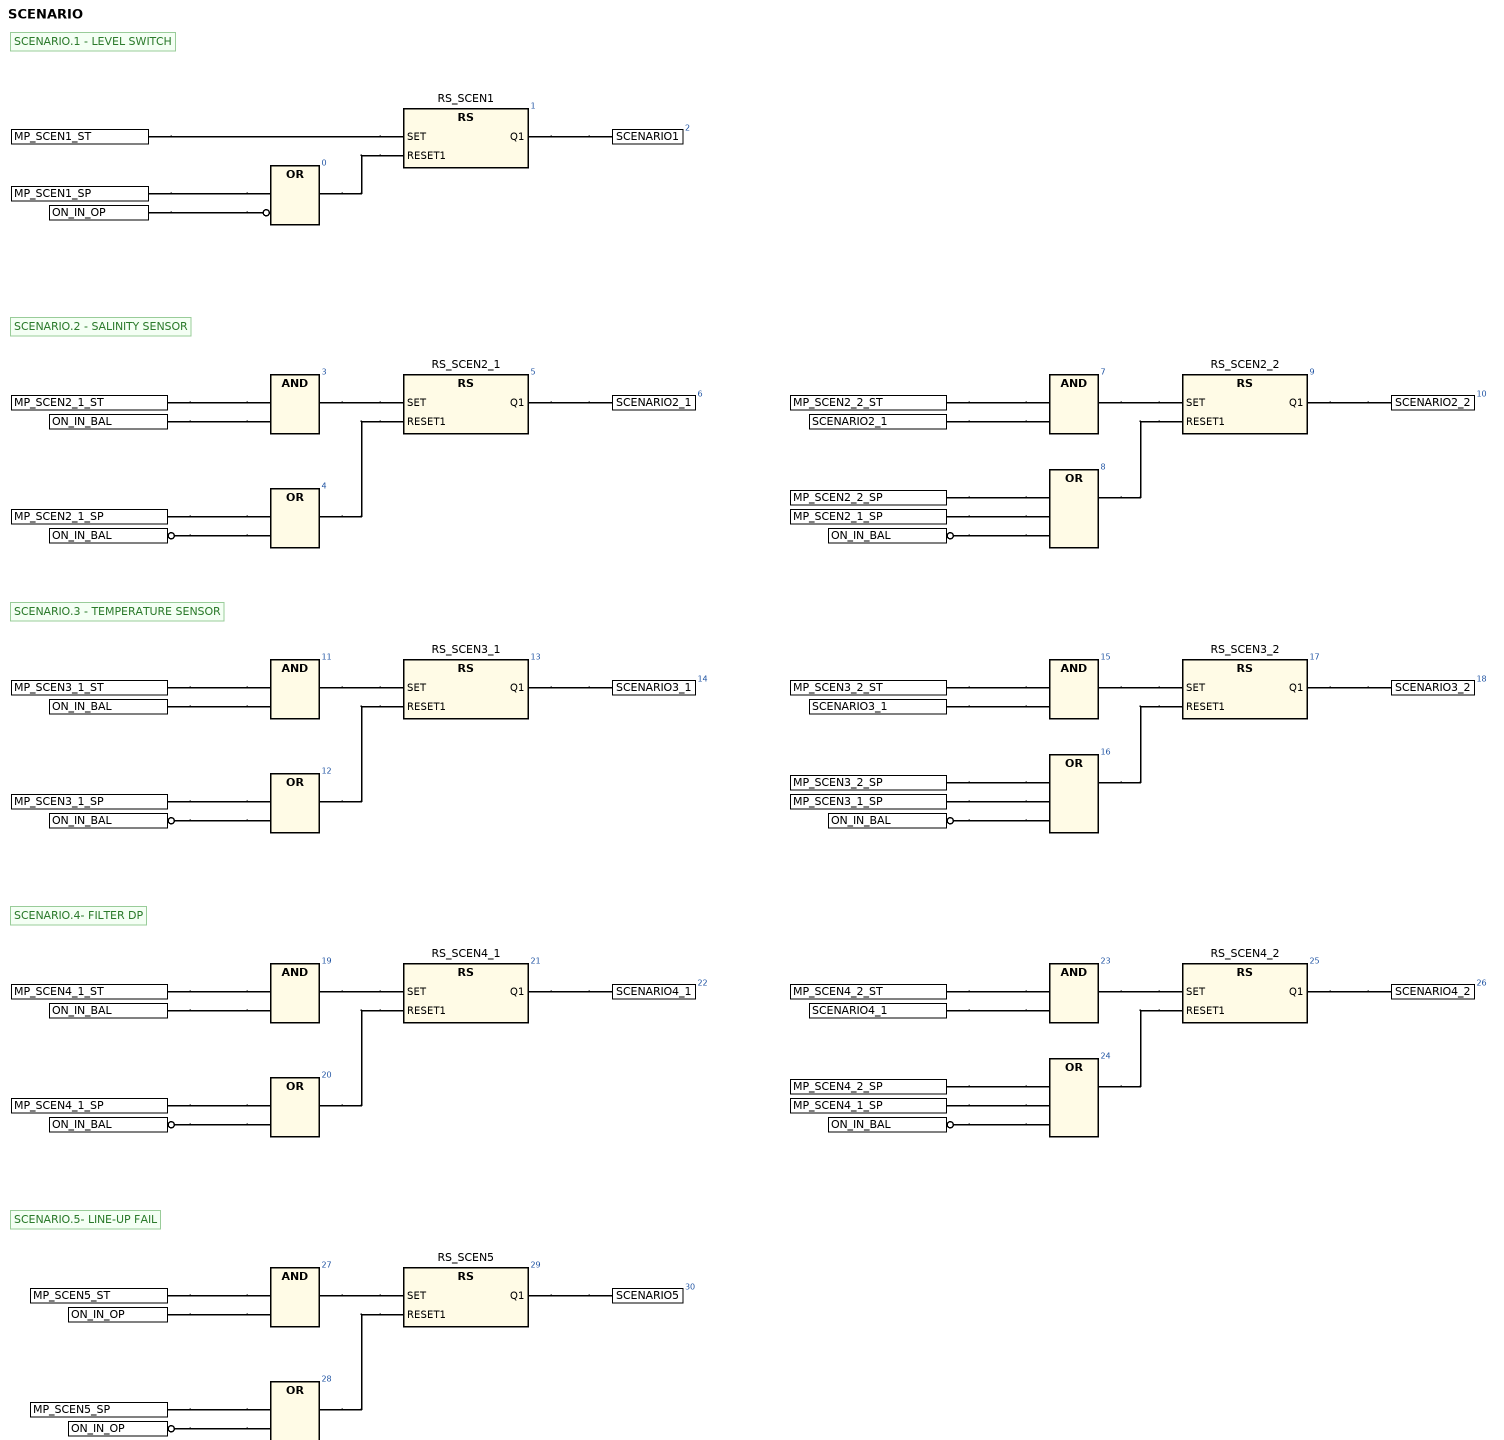
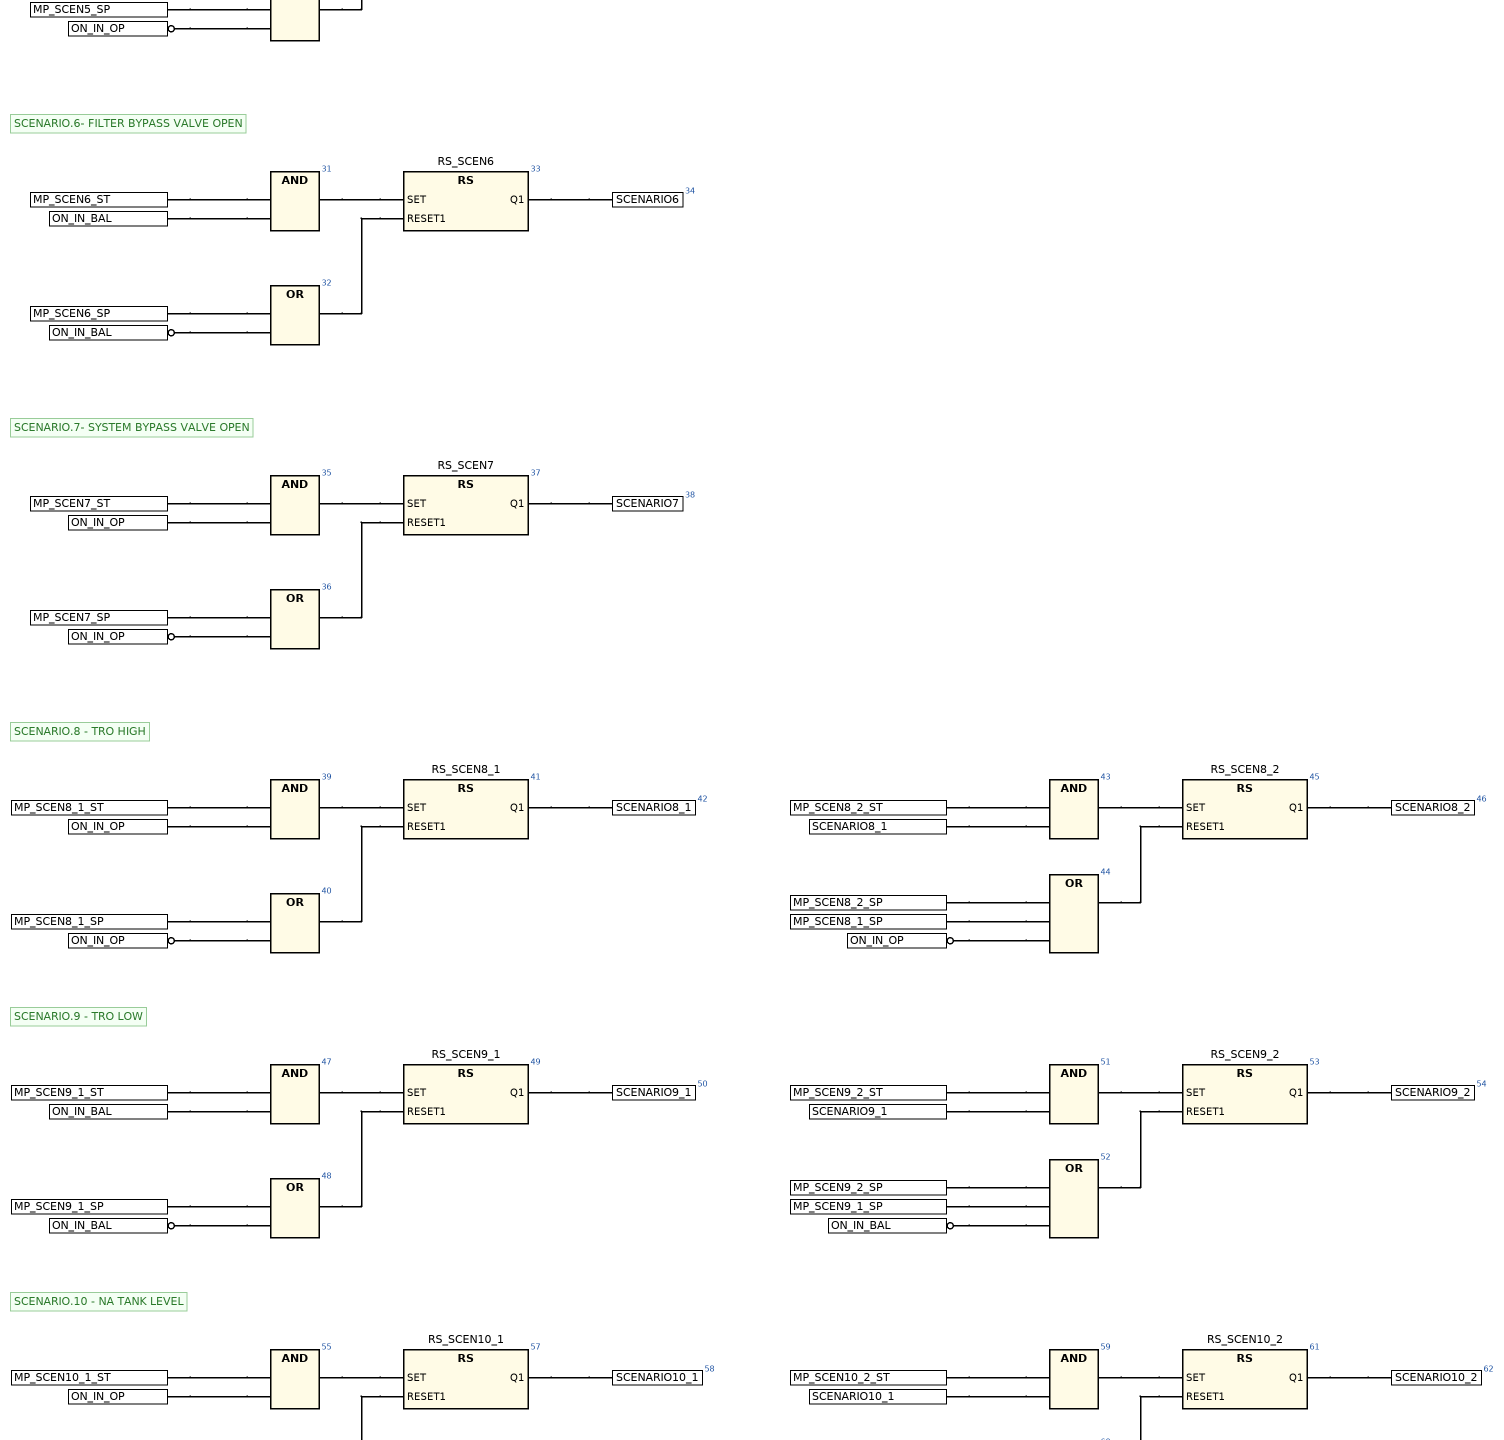
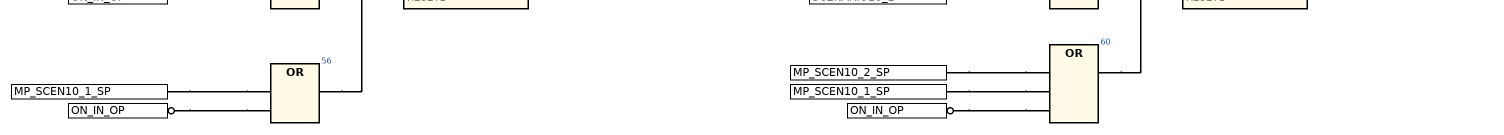
// SCENARIO.1 - LEVEL SWITCH
RS_SCEN1(SET := MP_SCEN1_ST, RESET1 := MP_SCEN1_SP OR NOT ON_IN_OP); // RS
SCENARIO1 := RS_SCEN1.Q1;
// SCENARIO.2 - SALINITY SENSOR
RS_SCEN2_1(SET := MP_SCEN2_1_ST AND ON_IN_BAL, RESET1 := MP_SCEN2_1_SP OR NOT ON_IN_BAL); // RS
SCENARIO2_1 := RS_SCEN2_1.Q1;
RS_SCEN2_2(SET := MP_SCEN2_2_ST AND SCENARIO2_1, RESET1 := MP_SCEN2_2_SP OR MP_SCEN2_1_SP OR NOT ON_IN_BAL); // RS
SCENARIO2_2 := RS_SCEN2_2.Q1;
// SCENARIO.3 - TEMPERATURE SENSOR
RS_SCEN3_1(SET := MP_SCEN3_1_ST AND ON_IN_BAL, RESET1 := MP_SCEN3_1_SP OR NOT ON_IN_BAL); // RS
SCENARIO3_1 := RS_SCEN3_1.Q1;
RS_SCEN3_2(SET := MP_SCEN3_2_ST AND SCENARIO3_1, RESET1 := MP_SCEN3_2_SP OR MP_SCEN3_1_SP OR NOT ON_IN_BAL); // RS
SCENARIO3_2 := RS_SCEN3_2.Q1;
// SCENARIO.4- FILTER DP
RS_SCEN4_1(SET := MP_SCEN4_1_ST AND ON_IN_BAL, RESET1 := MP_SCEN4_1_SP OR NOT ON_IN_BAL); // RS
SCENARIO4_1 := RS_SCEN4_1.Q1;
RS_SCEN4_2(SET := MP_SCEN4_2_ST AND SCENARIO4_1, RESET1 := MP_SCEN4_2_SP OR MP_SCEN4_1_SP OR NOT ON_IN_BAL); // RS
SCENARIO4_2 := RS_SCEN4_2.Q1;
// SCENARIO.5- LINE-UP FAIL
RS_SCEN5(SET := MP_SCEN5_ST AND ON_IN_OP, RESET1 := MP_SCEN5_SP OR NOT ON_IN_OP); // RS
SCENARIO5 := RS_SCEN5.Q1;
// SCENARIO.6- FILTER BYPASS VALVE OPEN
RS_SCEN6(SET := MP_SCEN6_ST AND ON_IN_BAL, RESET1 := MP_SCEN6_SP OR NOT ON_IN_BAL); // RS
SCENARIO6 := RS_SCEN6.Q1;
// SCENARIO.7- SYSTEM BYPASS VALVE OPEN
RS_SCEN7(SET := MP_SCEN7_ST AND ON_IN_OP, RESET1 := MP_SCEN7_SP OR NOT ON_IN_OP); // RS
SCENARIO7 := RS_SCEN7.Q1;
// SCENARIO.8 - TRO HIGH
RS_SCEN8_1(SET := MP_SCEN8_1_ST AND ON_IN_OP, RESET1 := MP_SCEN8_1_SP OR NOT ON_IN_OP); // RS
SCENARIO8_1 := RS_SCEN8_1.Q1;
RS_SCEN8_2(SET := MP_SCEN8_2_ST AND SCENARIO8_1, RESET1 := MP_SCEN8_2_SP OR MP_SCEN8_1_SP OR NOT ON_IN_OP); // RS
SCENARIO8_2 := RS_SCEN8_2.Q1;
// SCENARIO.9 - TRO LOW
RS_SCEN9_1(SET := MP_SCEN9_1_ST AND ON_IN_BAL, RESET1 := MP_SCEN9_1_SP OR NOT ON_IN_BAL); // RS
SCENARIO9_1 := RS_SCEN9_1.Q1;
RS_SCEN9_2(SET := MP_SCEN9_2_ST AND SCENARIO9_1, RESET1 := MP_SCEN9_2_SP OR MP_SCEN9_1_SP OR NOT ON_IN_BAL); // RS
SCENARIO9_2 := RS_SCEN9_2.Q1;
// SCENARIO.10 - NA TANK LEVEL
RS_SCEN10_1(SET := MP_SCEN10_1_ST AND ON_IN_OP, RESET1 := MP_SCEN10_1_SP OR NOT ON_IN_OP); // RS
SCENARIO10_1 := RS_SCEN10_1.Q1;
RS_SCEN10_2(SET := MP_SCEN10_2_ST AND SCENARIO10_1, RESET1 := MP_SCEN10_2_SP OR MP_SCEN10_1_SP OR NOT ON_IN_OP); // RS
SCENARIO10_2 := RS_SCEN10_2.Q1;

END_PROGRAM

// Device/Application/Logic/0.SIMULATION/SIMULATION_CAL
PROGRAM SIMULATION_CAL
VAR
	SM_RF_TRO_0: SM_RF_TRO;
END_VAR
VAR // added by the converter: edge detectors and wires of the graphical bodies
    _w1, _w2, _w3, _w4, _w5, _w6, _w7 : ANY;
END_VAR

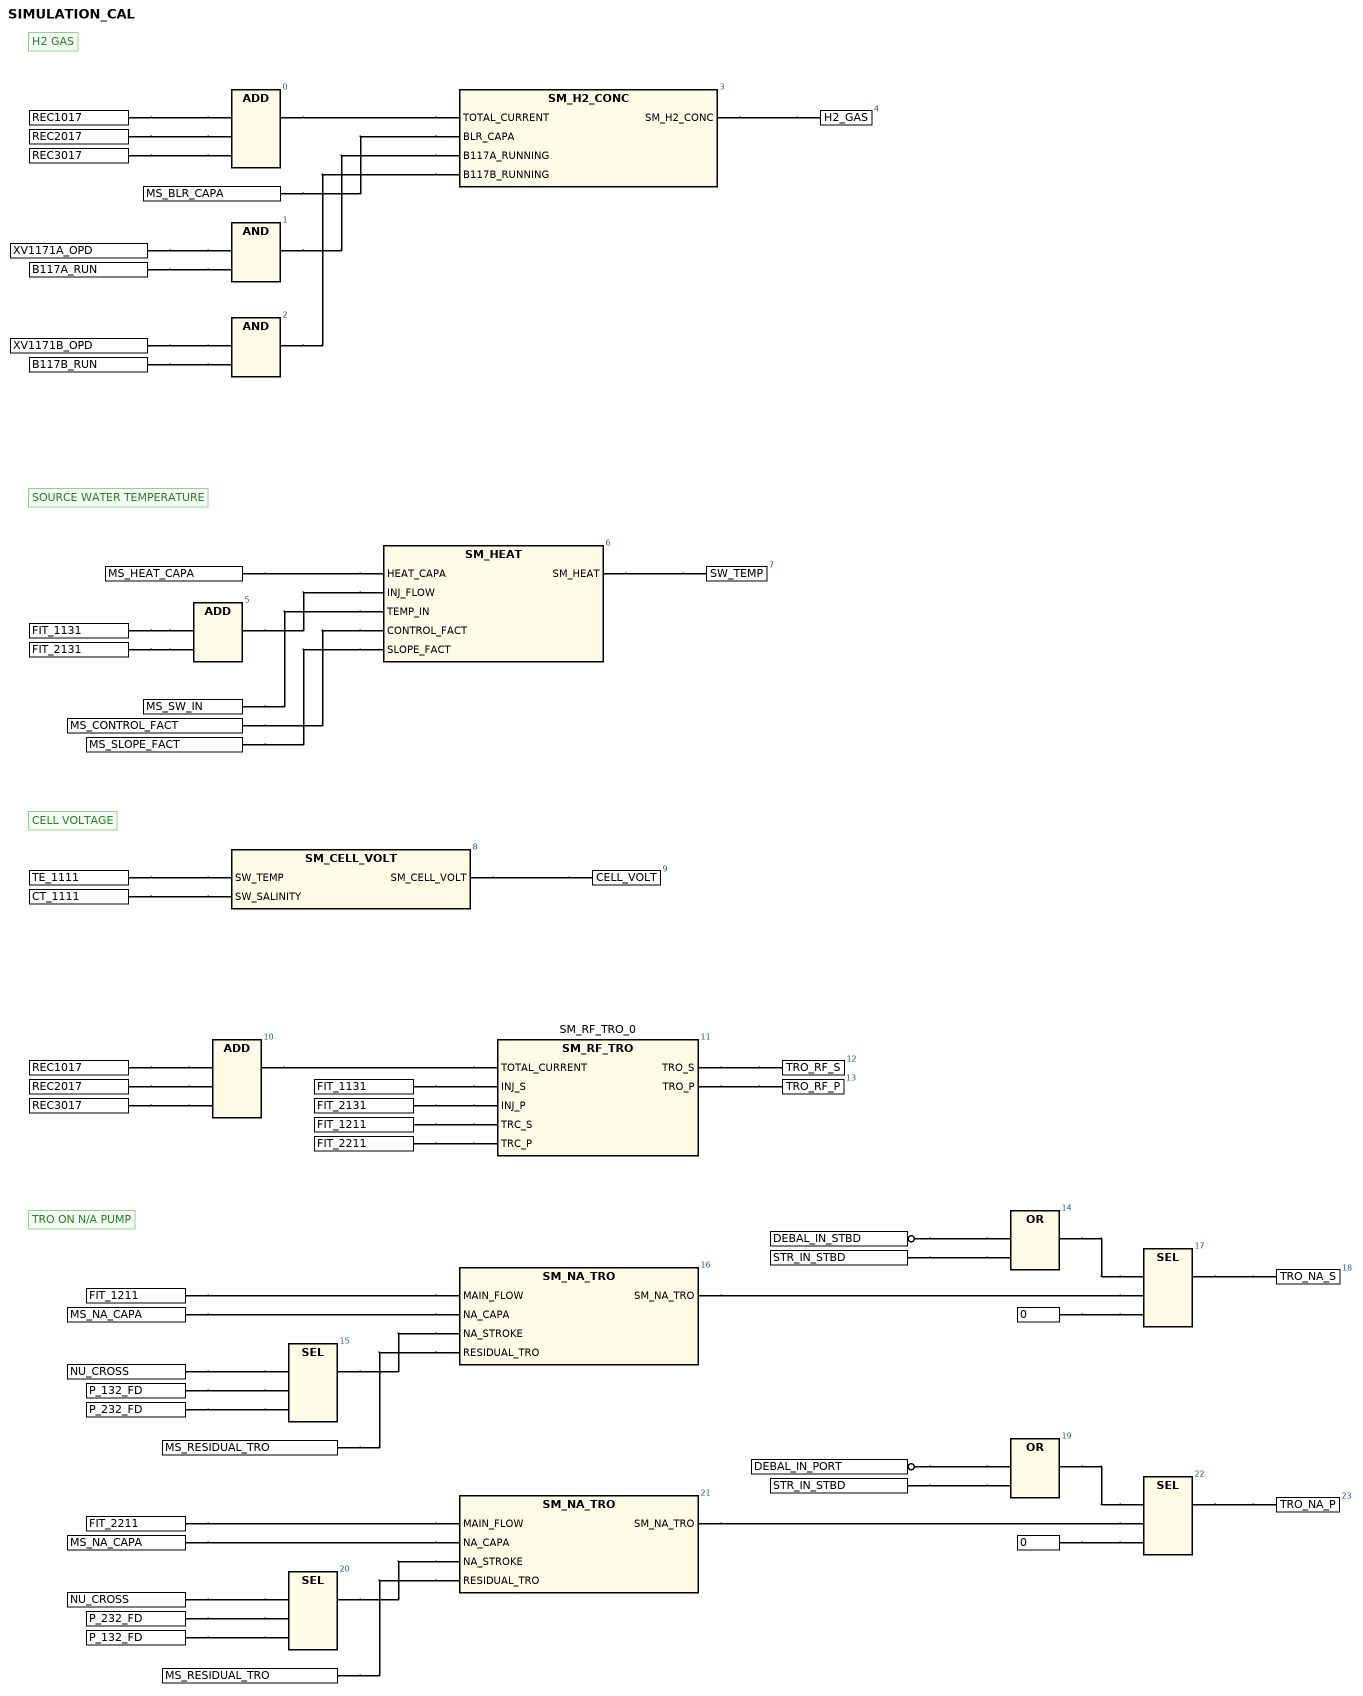
// H2 GAS
_w1 := SM_H2_CONC(TOTAL_CURRENT := REC1017 + REC2017 + REC3017, BLR_CAPA := MS_BLR_CAPA, B117A_RUNNING := XV1171A_OPD AND B117A_RUN, B117B_RUNNING := XV1171B_OPD AND B117B_RUN);
H2_GAS := _w1;
// SOURCE WATER TEMPERATURE
_w2 := SM_HEAT(HEAT_CAPA := MS_HEAT_CAPA, INJ_FLOW := FIT_1131 + FIT_2131, TEMP_IN := MS_SW_IN, CONTROL_FACT := MS_CONTROL_FACT, SLOPE_FACT := MS_SLOPE_FACT);
SW_TEMP := _w2;
// CELL VOLTAGE
_w3 := SM_CELL_VOLT(SW_TEMP := TE_1111, SW_SALINITY := CT_1111);
CELL_VOLT := _w3;
SM_RF_TRO_0(
    TOTAL_CURRENT := REC1017 + REC2017 + REC3017,
    INJ_S := FIT_1131,
    INJ_P := FIT_2131,
    TRC_S := FIT_1211,
    TRC_P := FIT_2211); // SM_RF_TRO
TRO_RF_S := SM_RF_TRO_0.TRO_S;
TRO_RF_P := SM_RF_TRO_0.TRO_P;
_w4 := NOT DEBAL_IN_STBD OR STR_IN_STBD;
// TRO ON N/A PUMP
_w5 := SM_NA_TRO(MAIN_FLOW := FIT_1211, NA_CAPA := MS_NA_CAPA, NA_STROKE := SEL(NU_CROSS, P_132_FD, P_232_FD), RESIDUAL_TRO := MS_RESIDUAL_TRO);
TRO_NA_S := SEL(_w4, _w5, 0);
_w6 := NOT DEBAL_IN_PORT OR STR_IN_STBD;
_w7 := SM_NA_TRO(MAIN_FLOW := FIT_2211, NA_CAPA := MS_NA_CAPA, NA_STROKE := SEL(NU_CROSS, P_232_FD, P_132_FD), RESIDUAL_TRO := MS_RESIDUAL_TRO);
TRO_NA_P := SEL(_w6, _w7, 0);

END_PROGRAM

// Device/Application/Logic/0.SIMULATION FBD/SM_H2_CONC
FUNCTION SM_H2_CONC : REAL
VAR_INPUT
	TOTAL_CURRENT : REAL;
	BLR_CAPA : REAL;
	B117A_RUNNING : BOOL;
	B117B_RUNNING : BOOL;
END_VAR
VAR
	CURR_T : REAL;					// CURRENT PER CELL
	FLOW_AIR : REAL;				// AIR FLOW
	FLOW_H2 : REAL;
	FLOW_T : REAL;
	CURR_EFF : REAL := 1;
	SEP_EFF : REAL := 0.7;
	CELL_N : REAL := 41;
	MWH2 : REAL := 2.01588;
	FARA : REAL := 96484.55461;
	H2_DEN : REAL := 0.08375;		// H2 DENSITY
	MASS_FLOW : REAL;
END_VAR

CURR_T := CELL_N * TOTAL_CURRENT;
MASS_FLOW := CURR_T / FARA / 2 *MWH2 * CURR_EFF / 1000 * 3600;
FLOW_AIR := SEL(B117A_RUNNING, 0, BLR_CAPA) + SEL(B117B_RUNNING, 0, BLR_CAPA); 
FLOW_H2 := MASS_FLOW / H2_DEN * SEP_EFF;
FLOW_T := FLOW_H2 + FLOW_AIR;

IF(FLOW_T =0) THEN
	SM_H2_CONC := 0;
ELSE
	SM_H2_CONC := FLOW_H2 / FLOW_T * 100;	
END_IF

END_FUNCTION

// Device/Application/Logic/0.SIMULATION FBD/SM_HEAT
FUNCTION SM_HEAT : REAL
VAR_INPUT
	HEAT_CAPA : REAL;
	INJ_FLOW : REAL;
	TEMP_IN : REAL;
	CONTROL_FACT : REAL;
	SLOPE_FACT : REAL;
END_VAR
VAR
	M : REAL;			// SLOPE
	K1 : REAL;
	Q1 : REAL;
	Q : REAL;
END_VAR

K1 := EXPT(CONTROL_FACT,INJ_FLOW/HEAT_CAPA);
M := SLOPE_FACT * HEAT_CAPA;
Q1 := M*(TEMP_IN - 35);
Q := Q1*K1;
IF(INJ_FLOW = 0) THEN
	SM_HEAT := TEMP_IN;
ELSE
	SM_HEAT := TEMP_IN + Q/(INJ_FLOW*4031);
END_IF

END_FUNCTION

// Device/Application/Logic/0.SIMULATION FBD/SM_CELL_VOLT
FUNCTION SM_CELL_VOLT : REAL
VAR_INPUT
	SW_TEMP : REAL;
	SW_SALINITY : REAL;
END_VAR
VAR
	a : LREAL := 2.15940688775066E-04;
	b : LREAL := 3.49304138321519E-06;
	c : LREAL := 9.41627678571512E-04;
	d : LREAL := 1.03922619047725E-06;
	e : LREAL := -4.8946513605481E-06;
	f : LREAL := 2.80843622448971E-05;
	g : LREAL := -1.78611111111348E-08;
	h : LREAL := 4.29841269841794E-08;
	i : LREAL := -9.80663265305954E-08;
	j : LREAL := 9.26111111111132E-08;
	X : LREAL;
END_VAR

X := (((((((((a + (b * SW_TEMP)) + (c * SW_SALINITY)) + (d * EXPT(SW_TEMP,2))) + (e * EXPT(SW_SALINITY,2))) + ((f * SW_TEMP) * SW_SALINITY)) + (g * EXPT(SW_TEMP,3)))
 + (h * EXPT(SW_SALINITY,3))) + ((i * SW_TEMP) * EXPT(SW_SALINITY,2))) + ((j * EXPT(SW_TEMP,2)) * SW_SALINITY));
SM_CELL_VOLT := 1.8 * EXPT(x,-0.18) * 41;

END_FUNCTION

// Device/Application/Logic/0.SIMULATION FBD/SM_RF_TRO
FUNCTION_BLOCK SM_RF_TRO
VAR_INPUT
	TOTAL_CURRENT : REAL;
	INJ_S : REAL;
	INJ_P : REAL;
	TRC_S : REAL;
	TRC_P : REAL;
END_VAR
VAR_OUTPUT
	TRO_S : REAL;
	TRO_P : REAL;
END_VAR
VAR
	CURR_EFF : REAL := 0.7;			//Current efficiency : 0~1
	FARA : REAL := 96484.55461;		//Faraday constant
	MWCL : REAL := 70.9054;			//M.W. of Chlorine
	CELL_N : REAL := 41;			//No. of cell 
	CURR_T : REAL;					//Total currunt
	CLPROD : REAL;
	INJ_RATIO_S : REAL;
	INJ_RATIO_P : REAL;
END_VAR

CURR_T := TOTAL_CURRENT * CELL_N;
CLPROD := CURR_T / FARA / 2 * MWCL * CURR_EFF / 1000 * 3600;

IF(INJ_S = 0 OR TRC_S = 0) THEN
	TRO_S := 0;
ELSE
	INJ_RATIO_S := INJ_S / (INJ_S + INJ_P);
	TRO_S := CLPROD * INJ_RATIO_S * 1000 / TRC_S;
END_IF

IF(INJ_P = 0 OR TRC_P = 0) THEN
	TRO_P := 0;
ELSE
	INJ_RATIO_P := INJ_P / (INJ_S + INJ_P);
	TRO_P := CLPROD * INJ_RATIO_P * 1000 / TRC_P;
END_IF

END_FUNCTION_BLOCK

// Device/Application/Logic/0.SIMULATION FBD/SM_NA_TRO
FUNCTION SM_NA_TRO : REAL
VAR_INPUT
	MAIN_FLOW : REAL;
	NA_CAPA : REAL;
	NA_STROKE : REAL;
	RESIDUAL_TRO : REAL;
END_VAR
VAR
	RESULT : REAL;
END_VAR

IF(MAIN_FLOW=0) THEN
	SM_NA_TRO := 0;
ELSE
	RESULT := RESIDUAL_TRO - (NA_CAPA * NA_STROKE / MAIN_FLOW * REAL#272.09);
	
	IF(RESULT < 0) THEN
		SM_NA_TRO := 0;
	ELSE
		SM_NA_TRO := RESULT;		
	END_IF
END_IF

END_FUNCTION

// Device/Application/Logic/0.SIMULATION/VIRTUAL_1
PROGRAM VIRTUAL_1
VAR
	SM_FOT_FIT1211: SM_FOT;
	SM_FOT_FIT2211: SM_FOT;
	SM_FOT_AIT151: SM_FOT;
	SM_FOT_AIT251: SM_FOT;
END_VAR
VAR // added by the converter: edge detectors and wires of the graphical bodies
    _w1, _w2, _w3, _w4, _w5, _w6, _w7, _w8, _w9, _w10, _w11, _w12, _w13, _w14, _w15, _w16, _w17, _w18 : ANY;
END_VAR

